LIN {X 0,Y 312.586,Z 149.548,A -85,B 0,C 180,E1 -15727.528,E2 -15727.528} C_VEL
LIN {X 0,Y 312.581,Z 149.547,A -85,B 0,C 180,E1 -15731.652,E2 -15731.652} C_VEL
LIN {X 0,Y 312.684,Z 149.533,A -85,B 0,C 180,E1 -15735.685,E2 -15735.685} C_VEL
LIN {X 0,Y 312.7,Z 149.532,A -85,B 0,C 180,E1 -15739.641,E2 -15739.641} C_VEL
LIN {X 0,Y 312.864,Z 149.511,A -85,B 0,C 180,E1 -15742.254,E2 -15742.254} C_VEL
LIN {X 0,Y 312.715,Z 149.533,A -85,B 0,C 180,E1 -15744.842,E2 -15744.842} C_VEL
LIN {X 0,Y 312.989,Z 149.499,A -85,B 0,C 180,E1 -15748.713,E2 -15748.713} C_VEL
LIN {X 0,Y 312.989,Z 149.496,A -85,B 0,C 180,E1 -15751.286,E2 -15751.286} C_VEL
LIN {X 0,Y 312.714,Z 149.531,A -85,B 0,C 180,E1 -15755.157,E2 -15755.157} C_VEL
LIN {X 0,Y 312.864,Z 149.51,A -85,B 0,C 180,E1 -15757.745,E2 -15757.745} C_VEL
LIN {X 0,Y 312.667,Z 149.535,A -85,B 0,C 180,E1 -15761.671,E2 -15761.671} C_VEL
LIN {X 0,Y 312.697,Z 149.533,A -85,B 0,C 180,E1 -15764.887,E2 -15764.887} C_VEL
LIN {X 0,Y 312.627,Z 149.54,A -85,B 0,C 180,E1 -15769.236,E2 -15769.236} C_VEL
LIN {X 0,Y 312.523,Z 149.554,A -85,B 0,C 180,E1 -15772.78,E2 -15772.78} C_VEL
LIN {X 0,Y 312.6,Z 149.546,A -85,B 0,C 180,E1 -15775.935,E2 -15775.935} C_VEL
LIN {X 0,Y 312.547,Z 149.551,A -85,B 0,C 180,E1 -15779.649,E2 -15779.649} C_VEL
LIN {X 0,Y 312.517,Z 149.556,A -85,B 0,C 180,E1 -15783.689,E2 -15783.689} C_VEL
LIN {X 0,Y 312.548,Z 149.55,A -85,B 0,C 180,E1 -15787.381,E2 -15787.381} C_VEL
LIN {X 0,Y 312.522,Z 149.553,A -85,B 0,C 180,E1 -15790.703,E2 -15790.703} C_VEL
LIN {X 0,Y 312.532,Z 149.554,A -85,B 0,C 180,E1 -15794.194,E2 -15794.194} C_VEL
LIN {X 0,Y 312.53,Z 149.556,A -85,B 0,C 180,E1 -15797.909,E2 -15797.909} C_VEL
LIN {X 0,Y 312.489,Z 149.557,A -85,B 0,C 180,E1 -15798.967,E2 -15798.967} C_VEL
LIN {X 0,Y 311.836,Z 149.643,A -85,B 0,C 180,E1 -15800.042,E2 -15800.042} C_VEL
LIN {X 0,Y 308.983,Z 149.998,A -85,B 0,C 180,E1 -15801.792,E2 -15801.792} C_VEL
LIN {X 0,Y 306.563,Z 150.296,A -85,B 0,C 180,E1 -15803.211,E2 -15803.211} C_VEL
LIN {X 0,Y 305.533,Z 150.424,A -85,B 0,C 180,E1 -15804.31,E2 -15804.31} C_VEL
LIN {X 0,Y 305.455,Z 150.433,A -85,B 0,C 180,E1 -15804.682,E2 -15804.682} C_VEL
LIN {X 0,Y 305.449,Z 150.434,A -85,B 0,C 180,E1 -15808.355,E2 -15808.355} C_VEL
LIN {X 0,Y 305.517,Z 150.427,A -85,B 0,C 180,E1 -15811.114,E2 -15811.114} C_VEL
LIN {X 0,Y 305.569,Z 150.42,A -85,B 0,C 180,E1 -15814.088,E2 -15814.088} C_VEL
LIN {X 0,Y 305.498,Z 150.428,A -85,B 0,C 180,E1 -15818.403,E2 -15818.403} C_VEL
LIN {X 0,Y 305.587,Z 150.421,A -85,B 0,C 180,E1 -15821.218,E2 -15821.218} C_VEL
LIN {X 0,Y 305.646,Z 150.413,A -85,B 0,C 180,E1 -15825.349,E2 -15825.349} C_VEL
LIN {X 0,Y 305.636,Z 150.413,A -85,B 0,C 180,E1 -15829.4,E2 -15829.4} C_VEL
LIN {X 0,Y 305.805,Z 150.39,A -85,B 0,C 180,E1 -15832.075,E2 -15832.075} C_VEL
LIN {X 0,Y 305.685,Z 150.407,A -85,B 0,C 180,E1 -15834.724,E2 -15834.724} C_VEL
LIN {X 0,Y 305.955,Z 150.374,A -85,B 0,C 180,E1 -15838.684,E2 -15838.684} C_VEL
LIN {X 0,Y 305.955,Z 150.372,A -85,B 0,C 180,E1 -15841.317,E2 -15841.317} C_VEL
LIN {X 0,Y 305.851,Z 150.388,A -85,B 0,C 180,E1 -15846.598,E2 -15846.598} C_VEL
LIN {X 0,Y 305.734,Z 150.399,A -85,B 0,C 180,E1 -15849.26,E2 -15849.26} C_VEL
LIN {X 0,Y 305.587,Z 150.417,A -85,B 0,C 180,E1 -15853.297,E2 -15853.297} C_VEL
LIN {X 0,Y 305.592,Z 150.418,A -85,B 0,C 180,E1 -15856.021,E2 -15856.021} C_VEL
LIN {X 0,Y 305.574,Z 150.418,A -85,B 0,C 180,E1 -15859.445,E2 -15859.445} C_VEL
LIN {X 0,Y 305.485,Z 150.43,A -85,B 0,C 180,E1 -15863.04,E2 -15863.04} C_VEL
LIN {X 0,Y 305.546,Z 150.427,A -85,B 0,C 180,E1 -15866.228,E2 -15866.228} C_VEL
LIN {X 0,Y 305.494,Z 150.428,A -85,B 0,C 180,E1 -15869.05,E2 -15869.05} C_VEL
LIN {X 0,Y 305.444,Z 150.438,A -85,B 0,C 180,E1 -15871.953,E2 -15871.953} C_VEL
LIN {X 0,Y 305.462,Z 150.432,A -85,B 0,C 180,E1 -15875.114,E2 -15875.114} C_VEL
LIN {X 0,Y 305.491,Z 150.43,A -85,B 0,C 180,E1 -15878.539,E2 -15878.539} C_VEL
LIN {X 0,Y 305.487,Z 150.43,A -85,B 0,C 180,E1 -15882.593,E2 -15882.593} C_VEL
LIN {X 0,Y 305.455,Z 150.435,A -85,B 0,C 180,E1 -15887.415,E2 -15887.415} C_VEL
LIN {X 0,Y 305.495,Z 150.432,A -85,B 0,C 180,E1 -15891.601,E2 -15891.601} C_VEL
LIN {X 0,Y 305.463,Z 150.433,A -85,B 0,C 180,E1 -15894.888,E2 -15894.888} C_VEL
LIN {X 0,Y 305.55,Z 150.588,A -85,B 0,C 180,E1 -15897.477,E2 -15897.477} C_VEL
LIN {X 0,Y 308.465,Z 164.645,A -85,B 0,C 180,E1 -15901.416,E2 -15901.416} C_VEL
LIN {X 0,Y 309.56,Z 170.48,A -85,B 0,C 180,E1 -15902.996,E2 -15902.996} C_VEL
LIN {X 0,Y 308.697,Z 179.088,A -85,B 0,C 180,E1 -15905.163,E2 -15905.163} C_VEL
LIN {X 0,Y 308.342,Z 181.983,A -85,B 0,C 180,E1 -15905.888,E2 -15905.888} C_VEL
LIN {X 0,Y 313.318,Z 226.374,A -85,B 0,C 180,E1 -15907.499,E2 -15907.499} C_VEL
LIN {X 0,Y 311.457,Z 291.139,A -85,B 0,C 180,E1 -15909.356,E2 -15909.356} C_VEL
LIN {X 0,Y 310.662,Z 304.701,A -85,B 0,C 180,E1 -15909.992,E2 -15909.992} C_VEL
LIN {X 0,Y 309.749,Z 316.693,A -85,B 0,C 180,E1 -15910.793,E2 -15910.793} C_VEL
LIN {X 0,Y 308.728,Z 327.693,A -85,B 0,C 180,E1 -15911.76,E2 -15911.76} C_VEL
LIN {X 0,Y 307.59,Z 339.295,A -85,B 0,C 180,E1 -15913.064,E2 -15913.064} C_VEL
LIN {X 0,Y 306.378,Z 350.376,A -85,B 0,C 180,E1 -15914.625,E2 -15914.625} C_VEL
LIN {X 0,Y 305.692,Z 358.469,A -85,B 0,C 180,E1 -15916.031,E2 -15916.031} C_VEL
LIN {X 0,Y 304.992,Z 366.419,A -85,B 0,C 180,E1 -15917.694,E2 -15917.694} C_VEL
LIN {X 0,Y 304.325,Z 374.155,A -85,B 0,C 180,E1 -15919.69,E2 -15919.69} C_VEL
LIN {X 0,Y 303.952,Z 381.267,A -85,B 0,C 180,E1 -15922.026,E2 -15922.026} C_VEL
LIN {X 0,Y 303.888,Z 385.785,A -85,B 0,C 180,E1 -15923.969,E2 -15923.969} C_VEL
LIN {X 0,Y 303.826,Z 389.338,A -85,B 0,C 180,E1 -15926.021,E2 -15926.021} C_VEL
LIN {X 0,Y 303.804,Z 391.012,A -85,B 0,C 180,E1 -15927.349,E2 -15927.349} C_VEL
LIN {X 0,Y 303.916,Z 392.26,A -85,B 0,C 180,E1 -15928.675,E2 -15928.675} C_VEL
LIN {X 0,Y 303.999,Z 393.067,A -85,B 0,C 180,E1 -15930,E2 -15930} C_VEL
LIN {X 0,Y 303.786,Z 393.382,A -85,B 0,C 180,E1 -15931.326,E2 -15931.326} C_VEL
LIN {X 0,Y 303.704,Z 393.287,A -85,B 0,C 180,E1 -15932.653,E2 -15932.653} C_VEL
LIN {X 0,Y 303.673,Z 392.784,A -85,B 0,C 180,E1 -15933.982,E2 -15933.982} C_VEL
LIN {X 0,Y 303.622,Z 391.636,A -85,B 0,C 180,E1 -15935.535,E2 -15935.535} C_VEL
LIN {X 0,Y 303.89,Z 388.673,A -85,B 0,C 180,E1 -15937.977,E2 -15937.977} C_VEL
LIN {X 0,Y 304.339,Z 385.131,A -85,B 0,C 180,E1 -15939.974,E2 -15939.974} C_VEL
LIN {X 0,Y 305.062,Z 380.498,A -85,B 0,C 180,E1 -15941.967,E2 -15941.967} C_VEL
LIN {X 0,Y 306.318,Z 374.653,A -85,B 0,C 180,E1 -15943.94,E2 -15943.94} C_VEL
LIN {X 0,Y 307.699,Z 367.423,A -85,B 0,C 180,E1 -15945.908,E2 -15945.908} C_VEL
LIN {X 0,Y 309.499,Z 358.5,A -85,B 0,C 180,E1 -15947.852,E2 -15947.852} C_VEL
LIN {X 0,Y 311.691,Z 348.451,A -85,B 0,C 180,E1 -15949.597,E2 -15949.597} C_VEL
LIN {X 0,Y 313.649,Z 338.405,A -85,B 0,C 180,E1 -15951.009,E2 -15951.009} C_VEL
LIN {X 0,Y 315.856,Z 325.87,A -85,B 0,C 180,E1 -15952.399,E2 -15952.399} C_VEL
LIN {X 0,Y 317.793,Z 313.439,A -85,B 0,C 180,E1 -15953.458,E2 -15953.458} C_VEL
LIN {X 0,Y 319.689,Z 299.024,A -85,B 0,C 180,E1 -15954.343,E2 -15954.343} C_VEL
LIN {X 0,Y 320.87,Z 286.162,A -85,B 0,C 180,E1 -15954.895,E2 -15954.895} C_VEL
LIN {X 0,Y 323.854,Z 227.495,A -85,B 0,C 180,E1 -15956.665,E2 -15956.665} C_VEL
LIN {X 0,Y 321.919,Z 211.124,A -85,B 0,C 180,E1 -15957.543,E2 -15957.543} C_VEL
LIN {X 0,Y 318.859,Z 193.947,A -85,B 0,C 180,E1 -15958.666,E2 -15958.666} C_VEL
LIN {X 0,Y 316.887,Z 185.521,A -85,B 0,C 180,E1 -15959.309,E2 -15959.309} C_VEL
LIN {X 0,Y 312.468,Z 176.034,A -85,B 0,C 180,E1 -15960.478,E2 -15960.478} C_VEL
LIN {X 0,Y 310.717,Z 168.166,A -85,B 0,C 180,E1 -15963.186,E2 -15963.186} C_VEL
LIN {X 0,Y 308.492,Z 160.006,A -85,B 0,C 180,E1 -15966.323,E2 -15966.323} C_VEL
LIN {X 0,Y 306.173,Z 152.7,A -85,B 0,C 180,E1 -15969.543,E2 -15969.543} C_VEL
LIN {X 0,Y 305.471,Z 150.434,A -85,B 0,C 180,E1 -15970.656,E2 -15970.656} C_VEL
LIN {X 0,Y 305.403,Z 150.44,A -85,B 0,C 180,E1 -15974.489,E2 -15974.489} C_VEL
LIN {X 0,Y 305.444,Z 150.431,A -85,B 0,C 180,E1 -15978.143,E2 -15978.143} C_VEL
LIN {X 0,Y 305.498,Z 150.424,A -85,B 0,C 180,E1 -15981.6,E2 -15981.6} C_VEL
LIN {X 0,Y 305.466,Z 150.431,A -85,B 0,C 180,E1 -15984.887,E2 -15984.887} C_VEL
LIN {X 0,Y 305.452,Z 150.428,A -85,B 0,C 180,E1 -15988.356,E2 -15988.356} C_VEL
LIN {X 0,Y 305.516,Z 150.423,A -85,B 0,C 180,E1 -15991.113,E2 -15991.113} C_VEL
LIN {X 0,Y 305.569,Z 150.415,A -85,B 0,C 180,E1 -15994.087,E2 -15994.087} C_VEL
LIN {X 0,Y 305.503,Z 150.431,A -85,B 0,C 180,E1 -15998.403,E2 -15998.403} C_VEL
LIN {X 0,Y 305.561,Z 150.421,A -85,B 0,C 180,E1 -16001.215,E2 -16001.215} C_VEL
LIN {X 0,Y 305.629,Z 150.415,A -85,B 0,C 180,E1 -16005.348,E2 -16005.348} C_VEL
LIN {X 0,Y 305.627,Z 150.415,A -85,B 0,C 180,E1 -16009.399,E2 -16009.399} C_VEL
LIN {X 0,Y 305.79,Z 150.494,A -85,B 0,C 180,E1 -16011.554,E2 -16011.554} C_VEL
LIN {X 0,Y 307.2,Z 154.947,A -85,B 0,C 180,E1 -16013.679,E2 -16013.679} C_VEL
LIN {X 0,Y 316.902,Z 170.364,A -85,B 0,C 180,E1 -16016.087,E2 -16016.087} C_VEL
LIN {X 0,Y 321.984,Z 179.999,A -85,B 0,C 180,E1 -16017.261,E2 -16017.261} C_VEL
LIN {X 0,Y 325.624,Z 188.448,A -85,B 0,C 180,E1 -16018.116,E2 -16018.116} C_VEL
LIN {X 0,Y 321.592,Z 261.751,A -85,B 0,C 180,E1 -16020.352,E2 -16020.352} C_VEL
LIN {X 0,Y 320.606,Z 274.961,A -85,B 0,C 180,E1 -16021.02,E2 -16021.02} C_VEL
LIN {X 0,Y 319.262,Z 287.316,A -85,B 0,C 180,E1 -16021.892,E2 -16021.892} C_VEL
LIN {X 0,Y 317.513,Z 299.966,A -85,B 0,C 180,E1 -16023.072,E2 -16023.072} C_VEL
LIN {X 0,Y 315.758,Z 310.435,A -85,B 0,C 180,E1 -16024.308,E2 -16024.308} C_VEL
LIN {X 0,Y 313.916,Z 320.373,A -85,B 0,C 180,E1 -16025.782,E2 -16025.782} C_VEL
LIN {X 0,Y 311.923,Z 329.891,A -85,B 0,C 180,E1 -16027.529,E2 -16027.529} C_VEL
LIN {X 0,Y 310.045,Z 338.248,A -85,B 0,C 180,E1 -16029.458,E2 -16029.458} C_VEL
LIN {X 0,Y 308.375,Z 345.16,A -85,B 0,C 180,E1 -16031.48,E2 -16031.48} C_VEL
LIN {X 0,Y 307.168,Z 349.957,A -85,B 0,C 180,E1 -16033.226,E2 -16033.226} C_VEL
LIN {X 0,Y 306.047,Z 354.407,A -85,B 0,C 180,E1 -16035.316,E2 -16035.316} C_VEL
LIN {X 0,Y 305.11,Z 357.667,A -85,B 0,C 180,E1 -16037.424,E2 -16037.424} C_VEL
LIN {X 0,Y 304.6,Z 359.297,A -85,B 0,C 180,E1 -16038.916,E2 -16038.916} C_VEL
LIN {X 0,Y 304.273,Z 360.262,A -85,B 0,C 180,E1 -16040.271,E2 -16040.271} C_VEL
LIN {X 0,Y 303.896,Z 360.929,A -85,B 0,C 180,E1 -16042.323,E2 -16042.323} C_VEL
LIN {X 0,Y 303.666,Z 360.491,A -85,B 0,C 180,E1 -16044.619,E2 -16044.619} C_VEL
LIN {X 0,Y 303.624,Z 359.576,A -85,B 0,C 180,E1 -16046.09,E2 -16046.09} C_VEL
LIN {X 0,Y 303.797,Z 356.925,A -85,B 0,C 180,E1 -16048.467,E2 -16048.467} C_VEL
LIN {X 0,Y 304.109,Z 353.399,A -85,B 0,C 180,E1 -16050.558,E2 -16050.558} C_VEL
LIN {X 0,Y 304.506,Z 348.138,A -85,B 0,C 180,E1 -16052.845,E2 -16052.845} C_VEL
LIN {X 0,Y 305.044,Z 342.283,A -85,B 0,C 180,E1 -16054.81,E2 -16054.81} C_VEL
LIN {X 0,Y 305.748,Z 335.246,A -85,B 0,C 180,E1 -16056.701,E2 -16056.701} C_VEL
LIN {X 0,Y 306.594,Z 326.786,A -85,B 0,C 180,E1 -16058.54,E2 -16058.54} C_VEL
LIN {X 0,Y 307.492,Z 317.339,A -85,B 0,C 180,E1 -16060.216,E2 -16060.216} C_VEL
LIN {X 0,Y 308.56,Z 306.406,A -85,B 0,C 180,E1 -16061.775,E2 -16061.775} C_VEL
LIN {X 0,Y 309.658,Z 293.744,A -85,B 0,C 180,E1 -16063.201,E2 -16063.201} C_VEL
LIN {X 0,Y 310.574,Z 280.985,A -85,B 0,C 180,E1 -16064.296,E2 -16064.296} C_VEL
LIN {X 0,Y 311.25,Z 267.383,A -85,B 0,C 180,E1 -16065.163,E2 -16065.163} C_VEL
LIN {X 0,Y 311.845,Z 253.446,A -85,B 0,C 180,E1 -16065.74,E2 -16065.74} C_VEL
LIN {X 0,Y 314.157,Z 176.783,A -85,B 0,C 180,E1 -16067.904,E2 -16067.904} C_VEL
LIN {X 0,Y 306.93,Z 154.768,A -85,B 0,C 180,E1 -16068.975,E2 -16068.975} C_VEL
LIN {X 0,Y 305.484,Z 150.432,A -85,B 0,C 180,E1 -16069.204,E2 -16069.204} C_VEL
LIN {X 0,Y 305.474,Z 150.434,A -85,B 0,C 180,E1 -16073.26,E2 -16073.26} C_VEL
LIN {X 0,Y 305.464,Z 150.432,A -85,B 0,C 180,E1 -16076.483,E2 -16076.483} C_VEL
LIN {X 0,Y 305.495,Z 150.43,A -85,B 0,C 180,E1 -16080.949,E2 -16080.949} C_VEL
LIN {X 0,Y 305.571,Z 150.419,A -85,B 0,C 180,E1 -16084.087,E2 -16084.087} C_VEL
LIN {X 0,Y 305.493,Z 150.429,A -85,B 0,C 180,E1 -16088.402,E2 -16088.402} C_VEL
LIN {X 0,Y 305.542,Z 150.428,A -85,B 0,C 180,E1 -16091.214,E2 -16091.214} C_VEL
LIN {X 0,Y 305.625,Z 150.415,A -85,B 0,C 180,E1 -16095.347,E2 -16095.347} C_VEL
LIN {X 0,Y 305.637,Z 150.413,A -85,B 0,C 180,E1 -16099.399,E2 -16099.399} C_VEL
LIN {X 0,Y 305.807,Z 150.389,A -85,B 0,C 180,E1 -16102.074,E2 -16102.074} C_VEL
LIN {X 0,Y 305.686,Z 150.408,A -85,B 0,C 180,E1 -16104.723,E2 -16104.723} C_VEL
LIN {X 0,Y 305.956,Z 150.375,A -85,B 0,C 180,E1 -16108.683,E2 -16108.683} C_VEL
LIN {X 0,Y 305.956,Z 150.372,A -85,B 0,C 180,E1 -16111.316,E2 -16111.316} C_VEL
LIN {X 0,Y 305.844,Z 150.39,A -85,B 0,C 180,E1 -16116.597,E2 -16116.597} C_VEL
LIN {X 0,Y 305.733,Z 150.399,A -85,B 0,C 180,E1 -16119.259,E2 -16119.259} C_VEL
LIN {X 0,Y 305.587,Z 150.417,A -85,B 0,C 180,E1 -16123.296,E2 -16123.296} C_VEL
LIN {X 0,Y 305.591,Z 150.418,A -85,B 0,C 180,E1 -16126.02,E2 -16126.02} C_VEL
LIN {X 0,Y 305.573,Z 150.418,A -85,B 0,C 180,E1 -16129.444,E2 -16129.444} C_VEL
LIN {X 0,Y 305.483,Z 150.43,A -85,B 0,C 180,E1 -16133.039,E2 -16133.039} C_VEL
LIN {X 0,Y 305.545,Z 150.427,A -85,B 0,C 180,E1 -16136.227,E2 -16136.227} C_VEL
LIN {X 0,Y 305.501,Z 150.427,A -85,B 0,C 180,E1 -16139.052,E2 -16139.052} C_VEL
LIN {X 0,Y 305.445,Z 150.438,A -85,B 0,C 180,E1 -16141.951,E2 -16141.951} C_VEL
LIN {X 0,Y 305.459,Z 150.432,A -85,B 0,C 180,E1 -16145.113,E2 -16145.113} C_VEL
LIN {X 0,Y 305.489,Z 150.43,A -85,B 0,C 180,E1 -16148.539,E2 -16148.539} C_VEL
LIN {X 0,Y 305.506,Z 150.427,A -85,B 0,C 180,E1 -16152.597,E2 -16152.597} C_VEL
LIN {X 0,Y 305.484,Z 150.431,A -85,B 0,C 180,E1 -16156.356,E2 -16156.356} C_VEL
LIN {X 0,Y 305.462,Z 150.436,A -85,B 0,C 180,E1 -16159.894,E2 -16159.894} C_VEL
LIN {X 0,Y 305.496,Z 150.433,A -85,B 0,C 180,E1 -16163.627,E2 -16163.627} C_VEL
LIN {X 0,Y 305.455,Z 150.433,A -85,B 0,C 180,E1 -16164.682,E2 -16164.682} C_VEL
LIN {X 0,Y 304.794,Z 150.519,A -85,B 0,C 180,E1 -16165.783,E2 -16165.783} C_VEL
LIN {X 0,Y 301.922,Z 150.879,A -85,B 0,C 180,E1 -16167.575,E2 -16167.575} C_VEL
LIN {X 0,Y 299.5,Z 151.177,A -85,B 0,C 180,E1 -16169.028,E2 -16169.028} C_VEL
LIN {X 0,Y 298.49,Z 151.302,A -85,B 0,C 180,E1 -16170.154,E2 -16170.154} C_VEL
LIN {X 0,Y 298.425,Z 151.308,A -85,B 0,C 180,E1 -16170.536,E2 -16170.536} C_VEL
LIN {X 0,Y 298.489,Z 151.306,A -85,B 0,C 180,E1 -16173.471,E2 -16173.471} C_VEL
LIN {X 0,Y 298.432,Z 151.309,A -85,B 0,C 180,E1 -16176.698,E2 -16176.698} C_VEL
LIN {X 0,Y 298.537,Z 151.296,A -85,B 0,C 180,E1 -16180.757,E2 -16180.757} C_VEL
LIN {X 0,Y 298.591,Z 151.292,A -85,B 0,C 180,E1 -16184.995,E2 -16184.995} C_VEL
LIN {X 0,Y 298.591,Z 151.293,A -85,B 0,C 180,E1 -16189.147,E2 -16189.147} C_VEL
LIN {X 0,Y 298.752,Z 151.268,A -85,B 0,C 180,E1 -16191.886,E2 -16191.886} C_VEL
LIN {X 0,Y 298.656,Z 151.282,A -85,B 0,C 180,E1 -16194.599,E2 -16194.599} C_VEL
LIN {X 0,Y 298.922,Z 151.25,A -85,B 0,C 180,E1 -16198.653,E2 -16198.653} C_VEL
LIN {X 0,Y 298.922,Z 151.248,A -85,B 0,C 180,E1 -16201.348,E2 -16201.348} C_VEL
LIN {X 0,Y 298.796,Z 151.268,A -85,B 0,C 180,E1 -16206.754,E2 -16206.754} C_VEL
LIN {X 0,Y 298.679,Z 151.278,A -85,B 0,C 180,E1 -16209.481,E2 -16209.481} C_VEL
LIN {X 0,Y 298.551,Z 151.293,A -85,B 0,C 180,E1 -16213.616,E2 -16213.616} C_VEL
LIN {X 0,Y 298.547,Z 151.298,A -85,B 0,C 180,E1 -16216.409,E2 -16216.409} C_VEL
LIN {X 0,Y 298.509,Z 151.298,A -85,B 0,C 180,E1 -16219.655,E2 -16219.655} C_VEL
LIN {X 0,Y 298.427,Z 151.309,A -85,B 0,C 180,E1 -16223.601,E2 -16223.601} C_VEL
LIN {X 0,Y 298.488,Z 151.304,A -85,B 0,C 180,E1 -16226.575,E2 -16226.575} C_VEL
LIN {X 0,Y 298.42,Z 151.31,A -85,B 0,C 180,E1 -16229.642,E2 -16229.642} C_VEL
LIN {X 0,Y 298.395,Z 151.314,A -85,B 0,C 180,E1 -16232.801,E2 -16232.801} C_VEL
LIN {X 0,Y 298.47,Z 151.303,A -85,B 0,C 180,E1 -16236.814,E2 -16236.814} C_VEL
LIN {X 0,Y 298.418,Z 151.31,A -85,B 0,C 180,E1 -16241.095,E2 -16241.095} C_VEL
LIN {X 0,Y 298.426,Z 151.309,A -85,B 0,C 180,E1 -16243.11,E2 -16243.11} C_VEL
LIN {X 0,Y 298.403,Z 151.312,A -85,B 0,C 180,E1 -16246.922,E2 -16246.922} C_VEL
LIN {X 0,Y 298.415,Z 151.311,A -85,B 0,C 180,E1 -16251.004,E2 -16251.004} C_VEL
LIN {X 0,Y 298.419,Z 151.314,A -85,B 0,C 180,E1 -16253.931,E2 -16253.931} C_VEL
LIN {X 0,Y 298.471,Z 151.352,A -85,B 0,C 180,E1 -16257.16,E2 -16257.16} C_VEL
LIN {X 0,Y 301.311,Z 164.922,A -85,B 0,C 180,E1 -16261.055,E2 -16261.055} C_VEL
LIN {X 0,Y 302.563,Z 172.208,A -85,B 0,C 180,E1 -16263.067,E2 -16263.067} C_VEL
LIN {X 0,Y 301.467,Z 181.646,A -85,B 0,C 180,E1 -16265.49,E2 -16265.49} C_VEL
LIN {X 0,Y 306.452,Z 226.423,A -85,B 0,C 180,E1 -16267.167,E2 -16267.167} C_VEL
LIN {X 0,Y 304.508,Z 291.26,A -85,B 0,C 180,E1 -16269.083,E2 -16269.083} C_VEL
LIN {X 0,Y 303.666,Z 305.37,A -85,B 0,C 180,E1 -16269.775,E2 -16269.775} C_VEL
LIN {X 0,Y 302.671,Z 318.042,A -85,B 0,C 180,E1 -16270.678,E2 -16270.678} C_VEL
LIN {X 0,Y 301.467,Z 330.243,A -85,B 0,C 180,E1 -16271.832,E2 -16271.832} C_VEL
LIN {X 0,Y 300.379,Z 341.324,A -85,B 0,C 180,E1 -16273.17,E2 -16273.17} C_VEL
LIN {X 0,Y 299.19,Z 351.635,A -85,B 0,C 180,E1 -16274.731,E2 -16274.731} C_VEL
LIN {X 0,Y 298.554,Z 358.819,A -85,B 0,C 180,E1 -16276.038,E2 -16276.038} C_VEL
LIN {X 0,Y 297.854,Z 366.641,A -85,B 0,C 180,E1 -16277.74,E2 -16277.74} C_VEL
LIN {X 0,Y 297.231,Z 374.28,A -85,B 0,C 180,E1 -16279.786,E2 -16279.786} C_VEL
LIN {X 0,Y 296.902,Z 380.38,A -85,B 0,C 180,E1 -16281.835,E2 -16281.835} C_VEL
LIN {X 0,Y 296.803,Z 385.375,A -85,B 0,C 180,E1 -16284.003,E2 -16284.003} C_VEL
LIN {X 0,Y 296.764,Z 388.686,A -85,B 0,C 180,E1 -16285.926,E2 -16285.926} C_VEL
LIN {X 0,Y 296.723,Z 390.414,A -85,B 0,C 180,E1 -16287.285,E2 -16287.285} C_VEL
LIN {X 0,Y 296.826,Z 391.706,A -85,B 0,C 180,E1 -16288.644,E2 -16288.644} C_VEL
LIN {X 0,Y 296.924,Z 392.569,A -85,B 0,C 180,E1 -16290.001,E2 -16290.001} C_VEL
LIN {X 0,Y 296.694,Z 392.955,A -85,B 0,C 180,E1 -16291.358,E2 -16291.358} C_VEL
LIN {X 0,Y 296.623,Z 392.901,A -85,B 0,C 180,E1 -16292.717,E2 -16292.717} C_VEL
LIN {X 0,Y 296.583,Z 392.441,A -85,B 0,C 180,E1 -16294.077,E2 -16294.077} C_VEL
LIN {X 0,Y 296.548,Z 391.522,A -85,B 0,C 180,E1 -16295.509,E2 -16295.509} C_VEL
LIN {X 0,Y 296.618,Z 390.264,A -85,B 0,C 180,E1 -16296.804,E2 -16296.804} C_VEL
LIN {X 0,Y 296.985,Z 387.5,A -85,B 0,C 180,E1 -16298.849,E2 -16298.849} C_VEL
LIN {X 0,Y 297.57,Z 383.699,A -85,B 0,C 180,E1 -16300.892,E2 -16300.892} C_VEL
LIN {X 0,Y 298.496,Z 378.775,A -85,B 0,C 180,E1 -16302.925,E2 -16302.925} C_VEL
LIN {X 0,Y 300.168,Z 371.468,A -85,B 0,C 180,E1 -16305.273,E2 -16305.273} C_VEL
LIN {X 0,Y 301.753,Z 363.674,A -85,B 0,C 180,E1 -16307.269,E2 -16307.269} C_VEL
LIN {X 0,Y 303.573,Z 355.722,A -85,B 0,C 180,E1 -16308.912,E2 -16308.912} C_VEL
LIN {X 0,Y 305.828,Z 345.069,A -85,B 0,C 180,E1 -16310.691,E2 -16310.691} C_VEL
LIN {X 0,Y 308.146,Z 334.358,A -85,B 0,C 180,E1 -16312.106,E2 -16312.106} C_VEL
LIN {X 0,Y 310.222,Z 322.647,A -85,B 0,C 180,E1 -16313.357,E2 -16313.357} C_VEL
LIN {X 0,Y 312.367,Z 309.416,A -85,B 0,C 180,E1 -16314.42,E2 -16314.42} C_VEL
LIN {X 0,Y 314.102,Z 295.961,A -85,B 0,C 180,E1 -16315.203,E2 -16315.203} C_VEL
LIN {X 0,Y 315.278,Z 281.766,A -85,B 0,C 180,E1 -16315.766,E2 -16315.766} C_VEL
LIN {X 0,Y 318.146,Z 228.588,A -85,B 0,C 180,E1 -16317.391,E2 -16317.391} C_VEL
LIN {X 0,Y 316.306,Z 212.407,A -85,B 0,C 180,E1 -16318.305,E2 -16318.305} C_VEL
LIN {X 0,Y 313.5,Z 196.283,A -85,B 0,C 180,E1 -16319.397,E2 -16319.397} C_VEL
LIN {X 0,Y 311.853,Z 189.166,A -85,B 0,C 180,E1 -16319.968,E2 -16319.968} C_VEL
LIN {X 0,Y 307.38,Z 179.825,A -85,B 0,C 180,E1 -16321.16,E2 -16321.16} C_VEL
LIN {X 0,Y 305.28,Z 175.365,A -85,B 0,C 180,E1 -16321.792,E2 -16321.792} C_VEL
LIN {X 0,Y 303.469,Z 167.901,A -85,B 0,C 180,E1 -16324.569,E2 -16324.569} C_VEL
LIN {X 0,Y 301.456,Z 160.696,A -85,B 0,C 180,E1 -16327.564,E2 -16327.564} C_VEL
LIN {X 0,Y 299.567,Z 154.906,A -85,B 0,C 180,E1 -16330.318,E2 -16330.318} C_VEL
LIN {X 0,Y 298.424,Z 151.31,A -85,B 0,C 180,E1 -16332.262,E2 -16332.262} C_VEL
LIN {X 0,Y 298.406,Z 151.311,A -85,B 0,C 180,E1 -16336.921,E2 -16336.921} C_VEL
LIN {X 0,Y 298.418,Z 151.303,A -85,B 0,C 180,E1 -16341.004,E2 -16341.004} C_VEL
LIN {X 0,Y 298.424,Z 151.303,A -85,B 0,C 180,E1 -16343.93,E2 -16343.93} C_VEL
LIN {X 0,Y 298.397,Z 151.309,A -85,B 0,C 180,E1 -16347.984,E2 -16347.984} C_VEL
LIN {X 0,Y 298.461,Z 151.302,A -85,B 0,C 180,E1 -16351.903,E2 -16351.903} C_VEL
LIN {X 0,Y 298.487,Z 151.3,A -85,B 0,C 180,E1 -16354.924,E2 -16354.924} C_VEL
LIN {X 0,Y 298.45,Z 151.303,A -85,B 0,C 180,E1 -16359.315,E2 -16359.315} C_VEL
LIN {X 0,Y 298.512,Z 151.295,A -85,B 0,C 180,E1 -16362.177,E2 -16362.177} C_VEL
LIN {X 0,Y 298.589,Z 151.288,A -85,B 0,C 180,E1 -16364.994,E2 -16364.994} C_VEL
LIN {X 0,Y 298.586,Z 151.29,A -85,B 0,C 180,E1 -16369.146,E2 -16369.146} C_VEL
LIN {X 0,Y 298.617,Z 151.462,A -85,B 0,C 180,E1 -16370.004,E2 -16370.004} C_VEL
LIN {X 0,Y 300.196,Z 155.742,A -85,B 0,C 180,E1 -16372.284,E2 -16372.284} C_VEL
LIN {X 0,Y 304.459,Z 162.336,A -85,B 0,C 180,E1 -16373.499,E2 -16373.499} C_VEL
LIN {X 0,Y 312.551,Z 175.162,A -85,B 0,C 180,E1 -16375.566,E2 -16375.566} C_VEL
LIN {X 0,Y 317.309,Z 184.427,A -85,B 0,C 180,E1 -16376.728,E2 -16376.728} C_VEL
LIN {X 0,Y 320.036,Z 190.794,A -85,B 0,C 180,E1 -16377.401,E2 -16377.401} C_VEL
LIN {X 0,Y 315.811,Z 261.792,A -85,B 0,C 180,E1 -16379.613,E2 -16379.613} C_VEL
LIN {X 0,Y 314.792,Z 274.33,A -85,B 0,C 180,E1 -16380.239,E2 -16380.239} C_VEL
LIN {X 0,Y 313.442,Z 286.936,A -85,B 0,C 180,E1 -16381.124,E2 -16381.124} C_VEL
LIN {X 0,Y 311.646,Z 299.174,A -85,B 0,C 180,E1 -16382.261,E2 -16382.261} C_VEL
LIN {X 0,Y 309.621,Z 310.675,A -85,B 0,C 180,E1 -16383.631,E2 -16383.631} C_VEL
LIN {X 0,Y 307.751,Z 320.284,A -85,B 0,C 180,E1 -16385.076,E2 -16385.076} C_VEL
LIN {X 0,Y 305.919,Z 328.628,A -85,B 0,C 180,E1 -16386.595,E2 -16386.595} C_VEL
LIN {X 0,Y 303.73,Z 337.727,A -85,B 0,C 180,E1 -16388.65,E2 -16388.65} C_VEL
LIN {X 0,Y 301.887,Z 344.926,A -85,B 0,C 180,E1 -16390.733,E2 -16390.733} C_VEL
LIN {X 0,Y 300.347,Z 350.607,A -85,B 0,C 180,E1 -16392.843,E2 -16392.843} C_VEL
LIN {X 0,Y 299.157,Z 354.976,A -85,B 0,C 180,E1 -16394.976,E2 -16394.976} C_VEL
LIN {X 0,Y 298.463,Z 357.275,A -85,B 0,C 180,E1 -16396.413,E2 -16396.413} C_VEL
LIN {X 0,Y 297.478,Z 360.119,A -85,B 0,C 180,E1 -16399.088,E2 -16399.088} C_VEL
LIN {X 0,Y 297.096,Z 361.081,A -85,B 0,C 180,E1 -16400.783,E2 -16400.783} C_VEL
LIN {X 0,Y 296.79,Z 361.374,A -85,B 0,C 180,E1 -16402.553,E2 -16402.553} C_VEL
LIN {X 0,Y 296.645,Z 361.183,A -85,B 0,C 180,E1 -16403.75,E2 -16403.75} C_VEL
LIN {X 0,Y 296.561,Z 360.099,A -85,B 0,C 180,E1 -16405.77,E2 -16405.77} C_VEL
LIN {X 0,Y 296.67,Z 357.453,A -85,B 0,C 180,E1 -16408.28,E2 -16408.28} C_VEL
LIN {X 0,Y 297.034,Z 353.67,A -85,B 0,C 180,E1 -16410.577,E2 -16410.577} C_VEL
LIN {X 0,Y 297.443,Z 348.367,A -85,B 0,C 180,E1 -16412.918,E2 -16412.918} C_VEL
LIN {X 0,Y 297.972,Z 342.594,A -85,B 0,C 180,E1 -16414.887,E2 -16414.887} C_VEL
LIN {X 0,Y 298.707,Z 335.306,A -85,B 0,C 180,E1 -16416.874,E2 -16416.874} C_VEL
LIN {X 0,Y 299.625,Z 326.238,A -85,B 0,C 180,E1 -16418.861,E2 -16418.861} C_VEL
LIN {X 0,Y 300.492,Z 317.509,A -85,B 0,C 180,E1 -16420.423,E2 -16420.423} C_VEL
LIN {X 0,Y 301.46,Z 308.031,A -85,B 0,C 180,E1 -16421.821,E2 -16421.821} C_VEL
LIN {X 0,Y 302.55,Z 295.876,A -85,B 0,C 180,E1 -16423.255,E2 -16423.255} C_VEL
LIN {X 0,Y 303.465,Z 284,A -85,B 0,C 180,E1 -16424.356,E2 -16424.356} C_VEL
LIN {X 0,Y 304.225,Z 270.889,A -85,B 0,C 180,E1 -16425.264,E2 -16425.264} C_VEL
LIN {X 0,Y 304.815,Z 256.905,A -85,B 0,C 180,E1 -16425.935,E2 -16425.935} C_VEL
LIN {X 0,Y 307.316,Z 177.999,A -85,B 0,C 180,E1 -16428.236,E2 -16428.236} C_VEL
LIN {X 0,Y 300.604,Z 157.594,A -85,B 0,C 180,E1 -16429.261,E2 -16429.261} C_VEL
LIN {X 0,Y 298.434,Z 151.313,A -85,B 0,C 180,E1 -16429.61,E2 -16429.61} C_VEL
LIN {X 0,Y 298.418,Z 151.313,A -85,B 0,C 180,E1 -16433.93,E2 -16433.93} C_VEL
LIN {X 0,Y 298.395,Z 151.315,A -85,B 0,C 180,E1 -16437.983,E2 -16437.983} C_VEL
LIN {X 0,Y 298.469,Z 151.306,A -85,B 0,C 180,E1 -16441.904,E2 -16441.904} C_VEL
LIN {X 0,Y 298.485,Z 151.304,A -85,B 0,C 180,E1 -16444.924,E2 -16444.924} C_VEL
LIN {X 0,Y 298.438,Z 151.312,A -85,B 0,C 180,E1 -16449.314,E2 -16449.314} C_VEL
LIN {X 0,Y 298.476,Z 151.303,A -85,B 0,C 180,E1 -16452.175,E2 -16452.175} C_VEL
LIN {X 0,Y 298.584,Z 151.293,A -85,B 0,C 180,E1 -16454.994,E2 -16454.994} C_VEL
LIN {X 0,Y 298.592,Z 151.293,A -85,B 0,C 180,E1 -16459.146,E2 -16459.146} C_VEL
LIN {X 0,Y 298.753,Z 151.268,A -85,B 0,C 180,E1 -16461.885,E2 -16461.885} C_VEL
LIN {X 0,Y 298.656,Z 151.282,A -85,B 0,C 180,E1 -16464.598,E2 -16464.598} C_VEL
LIN {X 0,Y 298.922,Z 151.251,A -85,B 0,C 180,E1 -16468.652,E2 -16468.652} C_VEL
LIN {X 0,Y 298.922,Z 151.248,A -85,B 0,C 180,E1 -16471.347,E2 -16471.347} C_VEL
LIN {X 0,Y 298.79,Z 151.268,A -85,B 0,C 180,E1 -16476.754,E2 -16476.754} C_VEL
LIN {X 0,Y 298.678,Z 151.277,A -85,B 0,C 180,E1 -16479.48,E2 -16479.48} C_VEL
LIN {X 0,Y 298.55,Z 151.293,A -85,B 0,C 180,E1 -16483.615,E2 -16483.615} C_VEL
LIN {X 0,Y 298.546,Z 151.299,A -85,B 0,C 180,E1 -16486.408,E2 -16486.408} C_VEL
LIN {X 0,Y 298.507,Z 151.298,A -85,B 0,C 180,E1 -16489.654,E2 -16489.654} C_VEL
LIN {X 0,Y 298.426,Z 151.309,A -85,B 0,C 180,E1 -16493.6,E2 -16493.6} C_VEL
LIN {X 0,Y 298.487,Z 151.303,A -85,B 0,C 180,E1 -16496.574,E2 -16496.574} C_VEL
LIN {X 0,Y 298.422,Z 151.31,A -85,B 0,C 180,E1 -16499.64,E2 -16499.64} C_VEL
LIN {X 0,Y 298.394,Z 151.313,A -85,B 0,C 180,E1 -16502.8,E2 -16502.8} C_VEL
LIN {X 0,Y 298.466,Z 151.304,A -85,B 0,C 180,E1 -16506.814,E2 -16506.814} C_VEL
LIN {X 0,Y 298.448,Z 151.307,A -85,B 0,C 180,E1 -16511.25,E2 -16511.25} C_VEL
LIN {X 0,Y 298.413,Z 151.31,A -85,B 0,C 180,E1 -16515.047,E2 -16515.047} C_VEL
LIN {X 0,Y 298.417,Z 151.31,A -85,B 0,C 180,E1 -16518.745,E2 -16518.745} C_VEL
LIN {X 0,Y 298.441,Z 151.307,A -85,B 0,C 180,E1 -16522.247,E2 -16522.247} C_VEL
LIN {X 0,Y 298.405,Z 151.316,A -85,B 0,C 180,E1 -16525.581,E2 -16525.581} C_VEL
LIN {X 0,Y 298.392,Z 151.313,A -85,B 0,C 180,E1 -16528.791,E2 -16528.791} C_VEL
LIN {X 0,Y 298.425,Z 151.308,A -85,B 0,C 180,E1 -16530.536,E2 -16530.536} C_VEL
LIN {X 0,Y 297.817,Z 151.388,A -85,B 0,C 180,E1 -16531.662,E2 -16531.662} C_VEL
LIN {X 0,Y 295.034,Z 151.736,A -85,B 0,C 180,E1 -16533.499,E2 -16533.499} C_VEL
LIN {X 0,Y 292.614,Z 152.035,A -85,B 0,C 180,E1 -16534.988,E2 -16534.988} C_VEL
LIN {X 0,Y 291.53,Z 152.169,A -85,B 0,C 180,E1 -16536.141,E2 -16536.141} C_VEL
LIN {X 0,Y 291.419,Z 152.182,A -85,B 0,C 180,E1 -16536.532,E2 -16536.532} C_VEL
LIN {X 0,Y 291.455,Z 152.177,A -85,B 0,C 180,E1 -16540.271,E2 -16540.271} C_VEL
LIN {X 0,Y 291.552,Z 152.166,A -85,B 0,C 180,E1 -16544.624,E2 -16544.624} C_VEL
LIN {X 0,Y 291.534,Z 152.17,A -85,B 0,C 180,E1 -16548.881,E2 -16548.881} C_VEL
LIN {X 0,Y 291.703,Z 152.147,A -85,B 0,C 180,E1 -16551.689,E2 -16551.689} C_VEL
LIN {X 0,Y 291.626,Z 152.157,A -85,B 0,C 180,E1 -16554.469,E2 -16554.469} C_VEL
LIN {X 0,Y 291.888,Z 152.126,A -85,B 0,C 180,E1 -16558.621,E2 -16558.621} C_VEL
LIN {X 0,Y 291.888,Z 152.124,A -85,B 0,C 180,E1 -16561.38,E2 -16561.38} C_VEL
LIN {X 0,Y 291.745,Z 152.145,A -85,B 0,C 180,E1 -16566.918,E2 -16566.918} C_VEL
LIN {X 0,Y 291.628,Z 152.156,A -85,B 0,C 180,E1 -16569.712,E2 -16569.712} C_VEL
LIN {X 0,Y 291.521,Z 152.169,A -85,B 0,C 180,E1 -16573.951,E2 -16573.951} C_VEL
LIN {X 0,Y 291.486,Z 152.176,A -85,B 0,C 180,E1 -16576.818,E2 -16576.818} C_VEL
LIN {X 0,Y 291.449,Z 152.178,A -85,B 0,C 180,E1 -16579.875,E2 -16579.875} C_VEL
LIN {X 0,Y 291.382,Z 152.19,A -85,B 0,C 180,E1 -16584.207,E2 -16584.207} C_VEL
LIN {X 0,Y 291.422,Z 152.181,A -85,B 0,C 180,E1 -16587.272,E2 -16587.272} C_VEL
LIN {X 0,Y 291.337,Z 152.195,A -85,B 0,C 180,E1 -16590.437,E2 -16590.437} C_VEL
LIN {X 0,Y 291.344,Z 152.193,A -85,B 0,C 180,E1 -16593.699,E2 -16593.699} C_VEL
LIN {X 0,Y 291.404,Z 152.183,A -85,B 0,C 180,E1 -16597.262,E2 -16597.262} C_VEL
LIN {X 0,Y 291.377,Z 152.188,A -85,B 0,C 180,E1 -16600.636,E2 -16600.636} C_VEL
LIN {X 0,Y 291.299,Z 152.197,A -85,B 0,C 180,E1 -16604.401,E2 -16604.401} C_VEL
LIN {X 0,Y 291.326,Z 152.195,A -85,B 0,C 180,E1 -16608.405,E2 -16608.405} C_VEL
LIN {X 0,Y 291.364,Z 152.19,A -85,B 0,C 180,E1 -16611.161,E2 -16611.161} C_VEL
LIN {X 0,Y 291.362,Z 152.19,A -85,B 0,C 180,E1 -16614.627,E2 -16614.627} C_VEL
LIN {X 0,Y 291.405,Z 152.279,A -85,B 0,C 180,E1 -16616.875,E2 -16616.875} C_VEL
LIN {X 0,Y 294.41,Z 166.621,A -85,B 0,C 180,E1 -16621.093,E2 -16621.093} C_VEL
LIN {X 0,Y 295.521,Z 172.532,A -85,B 0,C 180,E1 -16622.766,E2 -16622.766} C_VEL
LIN {X 0,Y 294.579,Z 181.534,A -85,B 0,C 180,E1 -16625.091,E2 -16625.091} C_VEL
LIN {X 0,Y 299.559,Z 227.691,A -85,B 0,C 180,E1 -16626.858,E2 -16626.858} C_VEL
LIN {X 0,Y 297.58,Z 291.39,A -85,B 0,C 180,E1 -16628.8,E2 -16628.8} C_VEL
LIN {X 0,Y 296.787,Z 304.621,A -85,B 0,C 180,E1 -16629.467,E2 -16629.467} C_VEL
LIN {X 0,Y 295.751,Z 317.396,A -85,B 0,C 180,E1 -16630.388,E2 -16630.388} C_VEL
LIN {X 0,Y 294.518,Z 329.644,A -85,B 0,C 180,E1 -16631.568,E2 -16631.568} C_VEL
LIN {X 0,Y 293.399,Z 340.773,A -85,B 0,C 180,E1 -16632.937,E2 -16632.937} C_VEL
LIN {X 0,Y 292.12,Z 351.812,A -85,B 0,C 180,E1 -16634.655,E2 -16634.655} C_VEL
LIN {X 0,Y 291.295,Z 360.841,A -85,B 0,C 180,E1 -16636.395,E2 -16636.395} C_VEL
LIN {X 0,Y 290.59,Z 368.262,A -85,B 0,C 180,E1 -16638.137,E2 -16638.137} C_VEL
LIN {X 0,Y 290.021,Z 375.495,A -85,B 0,C 180,E1 -16640.234,E2 -16640.234} C_VEL
LIN {X 0,Y 289.767,Z 381.234,A -85,B 0,C 180,E1 -16642.335,E2 -16642.335} C_VEL
LIN {X 0,Y 289.705,Z 385.676,A -85,B 0,C 180,E1 -16644.432,E2 -16644.432} C_VEL
LIN {X 0,Y 289.702,Z 387.989,A -85,B 0,C 180,E1 -16645.827,E2 -16645.827} C_VEL
LIN {X 0,Y 289.644,Z 389.804,A -85,B 0,C 180,E1 -16647.219,E2 -16647.219} C_VEL
LIN {X 0,Y 289.737,Z 391.138,A -85,B 0,C 180,E1 -16648.611,E2 -16648.611} C_VEL
LIN {X 0,Y 289.851,Z 392.046,A -85,B 0,C 180,E1 -16650.001,E2 -16650.001} C_VEL
LIN {X 0,Y 289.604,Z 392.506,A -85,B 0,C 180,E1 -16651.391,E2 -16651.391} C_VEL
LIN {X 0,Y 289.544,Z 392.517,A -85,B 0,C 180,E1 -16652.783,E2 -16652.783} C_VEL
LIN {X 0,Y 289.437,Z 391.397,A -85,B 0,C 180,E1 -16655.404,E2 -16655.404} C_VEL
LIN {X 0,Y 289.553,Z 390.051,A -85,B 0,C 180,E1 -16656.971,E2 -16656.971} C_VEL
LIN {X 0,Y 289.923,Z 387.362,A -85,B 0,C 180,E1 -16659.066,E2 -16659.066} C_VEL
LIN {X 0,Y 290.565,Z 383.674,A -85,B 0,C 180,E1 -16661.158,E2 -16661.158} C_VEL
LIN {X 0,Y 291.566,Z 378.898,A -85,B 0,C 180,E1 -16663.238,E2 -16663.238} C_VEL
LIN {X 0,Y 293.327,Z 371.748,A -85,B 0,C 180,E1 -16665.638,E2 -16665.638} C_VEL
LIN {X 0,Y 294.914,Z 364.443,A -85,B 0,C 180,E1 -16667.592,E2 -16667.592} C_VEL
LIN {X 0,Y 296.901,Z 356.311,A -85,B 0,C 180,E1 -16669.354,E2 -16669.354} C_VEL
LIN {X 0,Y 299.029,Z 347.079,A -85,B 0,C 180,E1 -16671.003,E2 -16671.003} C_VEL
LIN {X 0,Y 301.67,Z 335.665,A -85,B 0,C 180,E1 -16672.607,E2 -16672.607} C_VEL
LIN {X 0,Y 303.839,Z 324.392,A -85,B 0,C 180,E1 -16673.878,E2 -16673.878} C_VEL
LIN {X 0,Y 306.007,Z 311.87,A -85,B 0,C 180,E1 -16674.962,E2 -16674.962} C_VEL
LIN {X 0,Y 308.059,Z 297.428,A -85,B 0,C 180,E1 -16675.869,E2 -16675.869} C_VEL
LIN {X 0,Y 309.379,Z 283.198,A -85,B 0,C 180,E1 -16676.476,E2 -16676.476} C_VEL
LIN {X 0,Y 312.532,Z 229.371,A -85,B 0,C 180,E1 -16678.18,E2 -16678.18} C_VEL
LIN {X 0,Y 310.722,Z 213.529,A -85,B 0,C 180,E1 -16679.115,E2 -16679.115} C_VEL
LIN {X 0,Y 308.352,Z 199.12,A -85,B 0,C 180,E1 -16680.13,E2 -16680.13} C_VEL
LIN {X 0,Y 306.918,Z 192.788,A -85,B 0,C 180,E1 -16680.662,E2 -16680.662} C_VEL
LIN {X 0,Y 302.95,Z 184.33,A -85,B 0,C 180,E1 -16681.777,E2 -16681.777} C_VEL
LIN {X 0,Y 300.231,Z 179.012,A -85,B 0,C 180,E1 -16682.572,E2 -16682.572} C_VEL
LIN {X 0,Y 298.052,Z 174.602,A -85,B 0,C 180,E1 -16683.286,E2 -16683.286} C_VEL
LIN {X 0,Y 296.078,Z 166.936,A -85,B 0,C 180,E1 -16686.401,E2 -16686.401} C_VEL
LIN {X 0,Y 294.119,Z 160.44,A -85,B 0,C 180,E1 -16689.417,E2 -16689.417} C_VEL
LIN {X 0,Y 292.025,Z 154.353,A -85,B 0,C 180,E1 -16692.729,E2 -16692.729} C_VEL
LIN {X 0,Y 291.307,Z 152.195,A -85,B 0,C 180,E1 -16694.076,E2 -16694.076} C_VEL
LIN {X 0,Y 291.323,Z 152.195,A -85,B 0,C 180,E1 -16697.508,E2 -16697.508} C_VEL
LIN {X 0,Y 291.367,Z 152.181,A -85,B 0,C 180,E1 -16701.16,E2 -16701.16} C_VEL
LIN {X 0,Y 291.383,Z 152.185,A -85,B 0,C 180,E1 -16704.629,E2 -16704.629} C_VEL
LIN {X 0,Y 291.374,Z 152.184,A -85,B 0,C 180,E1 -16707.95,E2 -16707.95} C_VEL
LIN {X 0,Y 291.38,Z 152.183,A -85,B 0,C 180,E1 -16711.158,E2 -16711.158} C_VEL
LIN {X 0,Y 291.416,Z 152.178,A -85,B 0,C 180,E1 -16714.271,E2 -16714.271} C_VEL
LIN {X 0,Y 291.385,Z 152.183,A -85,B 0,C 180,E1 -16717.299,E2 -16717.299} C_VEL
LIN {X 0,Y 291.461,Z 152.175,A -85,B 0,C 180,E1 -16720.27,E2 -16720.27} C_VEL
LIN {X 0,Y 291.501,Z 152.17,A -85,B 0,C 180,E1 -16724.665,E2 -16724.665} C_VEL
LIN {X 0,Y 291.535,Z 152.322,A -85,B 0,C 180,E1 -16728.175,E2 -16728.175} C_VEL
LIN {X 0,Y 293.005,Z 156.516,A -85,B 0,C 180,E1 -16730.667,E2 -16730.667} C_VEL
LIN {X 0,Y 297.602,Z 162.945,A -85,B 0,C 180,E1 -16732.095,E2 -16732.095} C_VEL
LIN {X 0,Y 302.05,Z 169.865,A -85,B 0,C 180,E1 -16733.381,E2 -16733.381} C_VEL
LIN {X 0,Y 308.376,Z 180.311,A -85,B 0,C 180,E1 -16735.063,E2 -16735.063} C_VEL
LIN {X 0,Y 312.454,Z 188.42,A -85,B 0,C 180,E1 -16736.13,E2 -16736.13} C_VEL
LIN {X 0,Y 314.482,Z 193.12,A -85,B 0,C 180,E1 -16736.647,E2 -16736.647} C_VEL
LIN {X 0,Y 310.09,Z 262.242,A -85,B 0,C 180,E1 -16738.849,E2 -16738.849} C_VEL
LIN {X 0,Y 308.944,Z 275.275,A -85,B 0,C 180,E1 -16739.521,E2 -16739.521} C_VEL
LIN {X 0,Y 307.531,Z 287.536,A -85,B 0,C 180,E1 -16740.409,E2 -16740.409} C_VEL
LIN {X 0,Y 305.756,Z 299.005,A -85,B 0,C 180,E1 -16741.481,E2 -16741.481} C_VEL
LIN {X 0,Y 303.782,Z 309.929,A -85,B 0,C 180,E1 -16742.781,E2 -16742.781} C_VEL
LIN {X 0,Y 301.628,Z 320.38,A -85,B 0,C 180,E1 -16744.342,E2 -16744.342} C_VEL
LIN {X 0,Y 299.47,Z 329.569,A -85,B 0,C 180,E1 -16746.062,E2 -16746.062} C_VEL
LIN {X 0,Y 297.597,Z 336.876,A -85,B 0,C 180,E1 -16747.736,E2 -16747.736} C_VEL
LIN {X 0,Y 295.513,Z 344.591,A -85,B 0,C 180,E1 -16749.928,E2 -16749.928} C_VEL
LIN {X 0,Y 293.945,Z 350.077,A -85,B 0,C 180,E1 -16751.921,E2 -16751.921} C_VEL
LIN {X 0,Y 292.66,Z 354.329,A -85,B 0,C 180,E1 -16753.894,E2 -16753.894} C_VEL
LIN {X 0,Y 291.793,Z 357.055,A -85,B 0,C 180,E1 -16755.543,E2 -16755.543} C_VEL
LIN {X 0,Y 291.194,Z 358.762,A -85,B 0,C 180,E1 -16756.835,E2 -16756.835} C_VEL
LIN {X 0,Y 290.353,Z 360.927,A -85,B 0,C 180,E1 -16759.265,E2 -16759.265} C_VEL
LIN {X 0,Y 289.891,Z 361.74,A -85,B 0,C 180,E1 -16761.324,E2 -16761.324} C_VEL
LIN {X 0,Y 289.662,Z 361.742,A -85,B 0,C 180,E1 -16762.842,E2 -16762.842} C_VEL
LIN {X 0,Y 289.502,Z 361.254,A -85,B 0,C 180,E1 -16764.374,E2 -16764.374} C_VEL
LIN {X 0,Y 289.474,Z 360.131,A -85,B 0,C 180,E1 -16766.063,E2 -16766.063} C_VEL
LIN {X 0,Y 289.591,Z 357.737,A -85,B 0,C 180,E1 -16768.244,E2 -16768.244} C_VEL
LIN {X 0,Y 289.951,Z 353.898,A -85,B 0,C 180,E1 -16770.597,E2 -16770.597} C_VEL
LIN {X 0,Y 290.37,Z 348.539,A -85,B 0,C 180,E1 -16772.995,E2 -16772.995} C_VEL
LIN {X 0,Y 290.925,Z 342.639,A -85,B 0,C 180,E1 -16775.031,E2 -16775.031} C_VEL
LIN {X 0,Y 291.659,Z 335.36,A -85,B 0,C 180,E1 -16777.042,E2 -16777.042} C_VEL
LIN {X 0,Y 292.611,Z 326.228,A -85,B 0,C 180,E1 -16779.079,E2 -16779.079} C_VEL
LIN {X 0,Y 293.563,Z 317.163,A -85,B 0,C 180,E1 -16780.72,E2 -16780.72} C_VEL
LIN {X 0,Y 294.67,Z 306.188,A -85,B 0,C 180,E1 -16782.322,E2 -16782.322} C_VEL
LIN {X 0,Y 295.812,Z 293.704,A -85,B 0,C 180,E1 -16783.77,E2 -16783.77} C_VEL
LIN {X 0,Y 296.752,Z 280.809,A -85,B 0,C 180,E1 -16784.907,E2 -16784.907} C_VEL
LIN {X 0,Y 297.457,Z 267.609,A -85,B 0,C 180,E1 -16785.77,E2 -16785.77} C_VEL
LIN {X 0,Y 298.077,Z 253.321,A -85,B 0,C 180,E1 -16786.378,E2 -16786.378} C_VEL
LIN {X 0,Y 300.389,Z 178.97,A -85,B 0,C 180,E1 -16788.592,E2 -16788.592} C_VEL
LIN {X 0,Y 293.949,Z 159.621,A -85,B 0,C 180,E1 -16789.594,E2 -16789.594} C_VEL
LIN {X 0,Y 291.387,Z 152.189,A -85,B 0,C 180,E1 -16790.006,E2 -16790.006} C_VEL
LIN {X 0,Y 291.407,Z 152.184,A -85,B 0,C 180,E1 -16792.919,E2 -16792.919} C_VEL
LIN {X 0,Y 291.344,Z 152.192,A -85,B 0,C 180,E1 -16796.301,E2 -16796.301} C_VEL
LIN {X 0,Y 291.387,Z 152.187,A -85,B 0,C 180,E1 -16800.259,E2 -16800.259} C_VEL
LIN {X 0,Y 291.42,Z 152.182,A -85,B 0,C 180,E1 -16804.272,E2 -16804.272} C_VEL
LIN {X 0,Y 291.379,Z 152.192,A -85,B 0,C 180,E1 -16807.299,E2 -16807.299} C_VEL
LIN {X 0,Y 291.457,Z 152.177,A -85,B 0,C 180,E1 -16810.27,E2 -16810.27} C_VEL
LIN {X 0,Y 291.496,Z 152.173,A -85,B 0,C 180,E1 -16814.665,E2 -16814.665} C_VEL
LIN {X 0,Y 291.536,Z 152.171,A -85,B 0,C 180,E1 -16818.88,E2 -16818.88} C_VEL
LIN {X 0,Y 291.704,Z 152.147,A -85,B 0,C 180,E1 -16821.688,E2 -16821.688} C_VEL
LIN {X 0,Y 291.627,Z 152.157,A -85,B 0,C 180,E1 -16824.468,E2 -16824.468} C_VEL
LIN {X 0,Y 291.889,Z 152.127,A -85,B 0,C 180,E1 -16828.62,E2 -16828.62} C_VEL
LIN {X 0,Y 291.888,Z 152.124,A -85,B 0,C 180,E1 -16831.379,E2 -16831.379} C_VEL
LIN {X 0,Y 291.739,Z 152.145,A -85,B 0,C 180,E1 -16836.918,E2 -16836.918} C_VEL
LIN {X 0,Y 291.627,Z 152.156,A -85,B 0,C 180,E1 -16839.711,E2 -16839.711} C_VEL
LIN {X 0,Y 291.52,Z 152.17,A -85,B 0,C 180,E1 -16843.95,E2 -16843.95} C_VEL
LIN {X 0,Y 291.484,Z 152.176,A -85,B 0,C 180,E1 -16846.817,E2 -16846.817} C_VEL
LIN {X 0,Y 291.448,Z 152.179,A -85,B 0,C 180,E1 -16849.874,E2 -16849.874} C_VEL
LIN {X 0,Y 291.38,Z 152.191,A -85,B 0,C 180,E1 -16854.206,E2 -16854.206} C_VEL
LIN {X 0,Y 291.422,Z 152.181,A -85,B 0,C 180,E1 -16857.271,E2 -16857.271} C_VEL
LIN {X 0,Y 291.338,Z 152.195,A -85,B 0,C 180,E1 -16860.436,E2 -16860.436} C_VEL
LIN {X 0,Y 291.342,Z 152.193,A -85,B 0,C 180,E1 -16863.698,E2 -16863.698} C_VEL
LIN {X 0,Y 291.401,Z 152.184,A -85,B 0,C 180,E1 -16867.261,E2 -16867.261} C_VEL
LIN {X 0,Y 291.398,Z 152.185,A -85,B 0,C 180,E1 -16870.631,E2 -16870.631} C_VEL
LIN {X 0,Y 291.349,Z 152.191,A -85,B 0,C 180,E1 -16874.39,E2 -16874.39} C_VEL
LIN {X 0,Y 291.354,Z 152.191,A -85,B 0,C 180,E1 -16878.397,E2 -16878.397} C_VEL
LIN {X 0,Y 291.377,Z 152.188,A -85,B 0,C 180,E1 -16881.163,E2 -16881.163} C_VEL
LIN {X 0,Y 291.382,Z 152.186,A -85,B 0,C 180,E1 -16884.63,E2 -16884.63} C_VEL
LIN {X 0,Y 291.369,Z 152.19,A -85,B 0,C 180,E1 -16887.951,E2 -16887.951} C_VEL
LIN {X 0,Y 291.382,Z 152.188,A -85,B 0,C 180,E1 -16891.159,E2 -16891.159} C_VEL
LIN {X 0,Y 291.417,Z 152.182,A -85,B 0,C 180,E1 -16894.273,E2 -16894.273} C_VEL
LIN {X 0,Y 291.419,Z 152.182,A -85,B 0,C 180,E1 -16896.532,E2 -16896.532} C_VEL
LIN {X 0,Y 290.683,Z 152.277,A -85,B 0,C 180,E1 -16897.685,E2 -16897.685} C_VEL
LIN {X 0,Y 287.804,Z 152.634,A -85,B 0,C 180,E1 -16899.564,E2 -16899.564} C_VEL
LIN {X 0,Y 285.435,Z 152.93,A -85,B 0,C 180,E1 -16901.089,E2 -16901.089} C_VEL
LIN {X 0,Y 284.47,Z 153.047,A -85,B 0,C 180,E1 -16902.271,E2 -16902.271} C_VEL
LIN {X 0,Y 284.417,Z 153.055,A -85,B 0,C 180,E1 -16902.67,E2 -16902.67} C_VEL
LIN {X 0,Y 284.479,Z 153.047,A -85,B 0,C 180,E1 -16905.698,E2 -16905.698} C_VEL
LIN {X 0,Y 284.564,Z 153.036,A -85,B 0,C 180,E1 -16910.045,E2 -16910.045} C_VEL
LIN {X 0,Y 284.691,Z 153.024,A -85,B 0,C 180,E1 -16912.91,E2 -16912.91} C_VEL
LIN {X 0,Y 284.854,Z 153.002,A -85,B 0,C 180,E1 -16918.587,E2 -16918.587} C_VEL
LIN {X 0,Y 284.854,Z 153,A -85,B 0,C 180,E1 -16921.414,E2 -16921.414} C_VEL
LIN {X 0,Y 284.697,Z 153.021,A -85,B 0,C 180,E1 -16927.091,E2 -16927.091} C_VEL
LIN {X 0,Y 284.565,Z 153.036,A -85,B 0,C 180,E1 -16929.956,E2 -16929.956} C_VEL
LIN {X 0,Y 284.48,Z 153.048,A -85,B 0,C 180,E1 -16934.303,E2 -16934.303} C_VEL
LIN {X 0,Y 284.424,Z 153.053,A -85,B 0,C 180,E1 -16937.249,E2 -16937.249} C_VEL
LIN {X 0,Y 284.376,Z 153.062,A -85,B 0,C 180,E1 -16940.243,E2 -16940.243} C_VEL
LIN {X 0,Y 284.338,Z 153.065,A -85,B 0,C 180,E1 -16944.847,E2 -16944.847} C_VEL
LIN {X 0,Y 284.331,Z 153.067,A -85,B 0,C 180,E1 -16948.011,E2 -16948.011} C_VEL
LIN {X 0,Y 284.295,Z 153.069,A -85,B 0,C 180,E1 -16951.275,E2 -16951.275} C_VEL
LIN {X 0,Y 284.362,Z 153.061,A -85,B 0,C 180,E1 -16955.355,E2 -16955.355} C_VEL
LIN {X 0,Y 284.334,Z 153.068,A -85,B 0,C 180,E1 -16958.166,E2 -16958.166} C_VEL
LIN {X 0,Y 284.302,Z 153.073,A -85,B 0,C 180,E1 -16961.871,E2 -16961.871} C_VEL
LIN {X 0,Y 284.256,Z 153.077,A -85,B 0,C 180,E1 -16966.19,E2 -16966.19} C_VEL
LIN {X 0,Y 284.307,Z 153.071,A -85,B 0,C 180,E1 -16970.025,E2 -16970.025} C_VEL
LIN {X 0,Y 284.335,Z 153.07,A -85,B 0,C 180,E1 -16973.615,E2 -16973.615} C_VEL
LIN {X 0,Y 284.385,Z 153.189,A -85,B 0,C 180,E1 -16976.591,E2 -16976.591} C_VEL
LIN {X 0,Y 287.211,Z 166.814,A -85,B 0,C 180,E1 -16980.7,E2 -16980.7} C_VEL
LIN {X 0,Y 288.505,Z 174.149,A -85,B 0,C 180,E1 -16982.823,E2 -16982.823} C_VEL
LIN {X 0,Y 287.7,Z 181.099,A -85,B 0,C 180,E1 -16984.669,E2 -16984.669} C_VEL
LIN {X 0,Y 292.734,Z 226.959,A -85,B 0,C 180,E1 -16986.473,E2 -16986.473} C_VEL
LIN {X 0,Y 290.738,Z 290.445,A -85,B 0,C 180,E1 -16988.462,E2 -16988.462} C_VEL
LIN {X 0,Y 289.869,Z 303.747,A -85,B 0,C 180,E1 -16989.139,E2 -16989.139} C_VEL
LIN {X 0,Y 288.82,Z 316.65,A -85,B 0,C 180,E1 -16990.083,E2 -16990.083} C_VEL
LIN {X 0,Y 287.576,Z 328.945,A -85,B 0,C 180,E1 -16991.292,E2 -16991.292} C_VEL
LIN {X 0,Y 286.423,Z 340.122,A -85,B 0,C 180,E1 -16992.692,E2 -16992.692} C_VEL
LIN {X 0,Y 285.103,Z 351.202,A -85,B 0,C 180,E1 -16994.451,E2 -16994.451} C_VEL
LIN {X 0,Y 284.188,Z 361.095,A -85,B 0,C 180,E1 -16996.413,E2 -16996.413} C_VEL
LIN {X 0,Y 283.318,Z 369.657,A -85,B 0,C 180,E1 -16998.554,E2 -16998.554} C_VEL
LIN {X 0,Y 282.878,Z 376.54,A -85,B 0,C 180,E1 -17000.707,E2 -17000.707} C_VEL
LIN {X 0,Y 282.641,Z 381.978,A -85,B 0,C 180,E1 -17002.859,E2 -17002.859} C_VEL
LIN {X 0,Y 282.629,Z 386.148,A -85,B 0,C 180,E1 -17005.008,E2 -17005.008} C_VEL
LIN {X 0,Y 282.569,Z 389.15,A -85,B 0,C 180,E1 -17007.149,E2 -17007.149} C_VEL
LIN {X 0,Y 282.65,Z 390.559,A -85,B 0,C 180,E1 -17008.576,E2 -17008.576} C_VEL
LIN {X 0,Y 282.778,Z 391.518,A -85,B 0,C 180,E1 -17010.001,E2 -17010.001} C_VEL
LIN {X 0,Y 282.516,Z 392.026,A -85,B 0,C 180,E1 -17011.426,E2 -17011.426} C_VEL
LIN {X 0,Y 282.467,Z 392.128,A -85,B 0,C 180,E1 -17012.853,E2 -17012.853} C_VEL
LIN {X 0,Y 282.361,Z 391.221,A -85,B 0,C 180,E1 -17015.369,E2 -17015.369} C_VEL
LIN {X 0,Y 282.481,Z 389.817,A -85,B 0,C 180,E1 -17017.146,E2 -17017.146} C_VEL
LIN {X 0,Y 282.883,Z 387.242,A -85,B 0,C 180,E1 -17019.294,E2 -17019.294} C_VEL
LIN {X 0,Y 283.555,Z 383.662,A -85,B 0,C 180,E1 -17021.437,E2 -17021.437} C_VEL
LIN {X 0,Y 284.651,Z 378.997,A -85,B 0,C 180,E1 -17023.566,E2 -17023.566} C_VEL
LIN {X 0,Y 286.499,Z 372.036,A -85,B 0,C 180,E1 -17026.02,E2 -17026.02} C_VEL
LIN {X 0,Y 288.067,Z 365.342,A -85,B 0,C 180,E1 -17027.918,E2 -17027.918} C_VEL
LIN {X 0,Y 290.261,Z 357.026,A -85,B 0,C 180,E1 -17029.815,E2 -17029.815} C_VEL
LIN {X 0,Y 292.489,Z 347.996,A -85,B 0,C 180,E1 -17031.496,E2 -17031.496} C_VEL
LIN {X 0,Y 295.2,Z 336.973,A -85,B 0,C 180,E1 -17033.131,E2 -17033.131} C_VEL
LIN {X 0,Y 297.777,Z 324.554,A -85,B 0,C 180,E1 -17034.581,E2 -17034.581} C_VEL
LIN {X 0,Y 300.056,Z 312.388,A -85,B 0,C 180,E1 -17035.678,E2 -17035.678} C_VEL
LIN {X 0,Y 302.163,Z 298.433,A -85,B 0,C 180,E1 -17036.599,E2 -17036.599} C_VEL
LIN {X 0,Y 303.623,Z 285.304,A -85,B 0,C 180,E1 -17037.204,E2 -17037.204} C_VEL
LIN {X 0,Y 307.025,Z 230.877,A -85,B 0,C 180,E1 -17038.964,E2 -17038.964} C_VEL
LIN {X 0,Y 305.371,Z 215.387,A -85,B 0,C 180,E1 -17039.917,E2 -17039.917} C_VEL
LIN {X 0,Y 303.242,Z 201.67,A -85,B 0,C 180,E1 -17040.919,E2 -17040.919} C_VEL
LIN {X 0,Y 301.932,Z 196.07,A -85,B 0,C 180,E1 -17041.414,E2 -17041.414} C_VEL
LIN {X 0,Y 298.299,Z 188.202,A -85,B 0,C 180,E1 -17042.513,E2 -17042.513} C_VEL
LIN {X 0,Y 295.654,Z 183.064,A -85,B 0,C 180,E1 -17043.325,E2 -17043.325} C_VEL
LIN {X 0,Y 293.062,Z 178.27,A -85,B 0,C 180,E1 -17044.153,E2 -17044.153} C_VEL
LIN {X 0,Y 290.719,Z 173.805,A -85,B 0,C 180,E1 -17044.99,E2 -17044.99} C_VEL
LIN {X 0,Y 288.987,Z 167.269,A -85,B 0,C 180,E1 -17047.89,E2 -17047.89} C_VEL
LIN {X 0,Y 287.252,Z 161.816,A -85,B 0,C 180,E1 -17050.671,E2 -17050.671} C_VEL
LIN {X 0,Y 285.585,Z 156.926,A -85,B 0,C 180,E1 -17053.556,E2 -17053.556} C_VEL
LIN {X 0,Y 284.264,Z 153.07,A -85,B 0,C 180,E1 -17056.304,E2 -17056.304} C_VEL
LIN {X 0,Y 284.311,Z 153.065,A -85,B 0,C 180,E1 -17060.024,E2 -17060.024} C_VEL
LIN {X 0,Y 284.346,Z 153.055,A -85,B 0,C 180,E1 -17063.615,E2 -17063.615} C_VEL
LIN {X 0,Y 284.311,Z 153.067,A -85,B 0,C 180,E1 -17067.19,E2 -17067.19} C_VEL
LIN {X 0,Y 284.359,Z 153.063,A -85,B 0,C 180,E1 -17070.375,E2 -17070.375} C_VEL
LIN {X 0,Y 284.378,Z 153.057,A -85,B 0,C 180,E1 -17073.586,E2 -17073.586} C_VEL
LIN {X 0,Y 284.37,Z 153.056,A -85,B 0,C 180,E1 -17076.707,E2 -17076.707} C_VEL
LIN {X 0,Y 284.39,Z 153.057,A -85,B 0,C 180,E1 -17081.26,E2 -17081.26} C_VEL
LIN {X 0,Y 284.486,Z 153.078,A -85,B 0,C 180,E1 -17085.925,E2 -17085.925} C_VEL
LIN {X 0,Y 285.838,Z 157.286,A -85,B 0,C 180,E1 -17088.833,E2 -17088.833} C_VEL
LIN {X 0,Y 289.338,Z 161.911,A -85,B 0,C 180,E1 -17090.064,E2 -17090.064} C_VEL
LIN {X 0,Y 294.079,Z 168.576,A -85,B 0,C 180,E1 -17091.598,E2 -17091.598} C_VEL
LIN {X 0,Y 298.738,Z 176.141,A -85,B 0,C 180,E1 -17093.011,E2 -17093.011} C_VEL
LIN {X 0,Y 304.057,Z 185.069,A -85,B 0,C 180,E1 -17094.499,E2 -17094.499} C_VEL
LIN {X 0,Y 308.04,Z 193.204,A -85,B 0,C 180,E1 -17095.583,E2 -17095.583} C_VEL
LIN {X 0,Y 308.957,Z 195.331,A -85,B 0,C 180,E1 -17095.838,E2 -17095.838} C_VEL
LIN {X 0,Y 304.461,Z 262.962,A -85,B 0,C 180,E1 -17098.057,E2 -17098.057} C_VEL
LIN {X 0,Y 303.369,Z 274.844,A -85,B 0,C 180,E1 -17098.672,E2 -17098.672} C_VEL
LIN {X 0,Y 301.849,Z 287.601,A -85,B 0,C 180,E1 -17099.597,E2 -17099.597} C_VEL
LIN {X 0,Y 299.973,Z 298.978,A -85,B 0,C 180,E1 -17100.671,E2 -17100.671} C_VEL
LIN {X 0,Y 297.818,Z 310.192,A -85,B 0,C 180,E1 -17102.028,E2 -17102.028} C_VEL
LIN {X 0,Y 295.496,Z 320.768,A -85,B 0,C 180,E1 -17103.631,E2 -17103.631} C_VEL
LIN {X 0,Y 293.053,Z 330.567,A -85,B 0,C 180,E1 -17105.504,E2 -17105.504} C_VEL
LIN {X 0,Y 290.692,Z 339.209,A -85,B 0,C 180,E1 -17107.582,E2 -17107.582} C_VEL
LIN {X 0,Y 288.54,Z 346.426,A -85,B 0,C 180,E1 -17109.816,E2 -17109.816} C_VEL
LIN {X 0,Y 286.724,Z 352.17,A -85,B 0,C 180,E1 -17112.114,E2 -17112.114} C_VEL
LIN {X 0,Y 285.386,Z 356.243,A -85,B 0,C 180,E1 -17114.256,E2 -17114.256} C_VEL
LIN {X 0,Y 284.603,Z 358.427,A -85,B 0,C 180,E1 -17115.761,E2 -17115.761} C_VEL
LIN {X 0,Y 283.959,Z 360.095,A -85,B 0,C 180,E1 -17117.277,E2 -17117.277} C_VEL
LIN {X 0,Y 283.241,Z 361.645,A -85,B 0,C 180,E1 -17119.457,E2 -17119.457} C_VEL
LIN {X 0,Y 282.716,Z 362.222,A -85,B 0,C 180,E1 -17121.893,E2 -17121.893} C_VEL
LIN {X 0,Y 282.509,Z 361.969,A -85,B 0,C 180,E1 -17123.455,E2 -17123.455} C_VEL
LIN {X 0,Y 282.377,Z 361.171,A -85,B 0,C 180,E1 -17125.03,E2 -17125.03} C_VEL
LIN {X 0,Y 282.383,Z 359.89,A -85,B 0,C 180,E1 -17126.614,E2 -17126.614} C_VEL
LIN {X 0,Y 282.487,Z 358.017,A -85,B 0,C 180,E1 -17128.209,E2 -17128.209} C_VEL
LIN {X 0,Y 282.852,Z 354.119,A -85,B 0,C 180,E1 -17130.621,E2 -17130.621} C_VEL
LIN {X 0,Y 283.3,Z 348.691,A -85,B 0,C 180,E1 -17133.076,E2 -17133.076} C_VEL
LIN {X 0,Y 283.892,Z 342.518,A -85,B 0,C 180,E1 -17135.219,E2 -17135.219} C_VEL
LIN {X 0,Y 284.778,Z 334.003,A -85,B 0,C 180,E1 -17137.559,E2 -17137.559} C_VEL
LIN {X 0,Y 285.74,Z 325.021,A -85,B 0,C 180,E1 -17139.524,E2 -17139.524} C_VEL
LIN {X 0,Y 286.866,Z 314.271,A -85,B 0,C 180,E1 -17141.412,E2 -17141.412} C_VEL
LIN {X 0,Y 287.995,Z 303.415,A -85,B 0,C 180,E1 -17142.937,E2 -17142.937} C_VEL
LIN {X 0,Y 289.063,Z 290.684,A -85,B 0,C 180,E1 -17144.346,E2 -17144.346} C_VEL
LIN {X 0,Y 289.963,Z 279.04,A -85,B 0,C 180,E1 -17145.34,E2 -17145.34} C_VEL
LIN {X 0,Y 290.673,Z 265.528,A -85,B 0,C 180,E1 -17146.185,E2 -17146.185} C_VEL
LIN {X 0,Y 291.272,Z 251.705,A -85,B 0,C 180,E1 -17146.75,E2 -17146.75} C_VEL
LIN {X 0,Y 293.552,Z 180.316,A -85,B 0,C 180,E1 -17148.943,E2 -17148.943} C_VEL
LIN {X 0,Y 287.659,Z 162.583,A -85,B 0,C 180,E1 -17149.88,E2 -17149.88} C_VEL
LIN {X 0,Y 284.357,Z 153.063,A -85,B 0,C 180,E1 -17150.431,E2 -17150.431} C_VEL
LIN {X 0,Y 284.34,Z 153.064,A -85,B 0,C 180,E1 -17154.651,E2 -17154.651} C_VEL
LIN {X 0,Y 284.295,Z 153.07,A -85,B 0,C 180,E1 -17158.725,E2 -17158.725} C_VEL
LIN {X 0,Y 284.399,Z 153.059,A -85,B 0,C 180,E1 -17162.825,E2 -17162.825} C_VEL
LIN {X 0,Y 284.365,Z 153.062,A -85,B 0,C 180,E1 -17166.706,E2 -17166.706} C_VEL
LIN {X 0,Y 284.368,Z 153.065,A -85,B 0,C 180,E1 -17171.259,E2 -17171.259} C_VEL
LIN {X 0,Y 284.462,Z 153.048,A -85,B 0,C 180,E1 -17175.696,E2 -17175.696} C_VEL
LIN {X 0,Y 284.565,Z 153.036,A -85,B 0,C 180,E1 -17180.044,E2 -17180.044} C_VEL
LIN {X 0,Y 284.692,Z 153.024,A -85,B 0,C 180,E1 -17182.909,E2 -17182.909} C_VEL
LIN {X 0,Y 284.854,Z 153.002,A -85,B 0,C 180,E1 -17188.586,E2 -17188.586} C_VEL
LIN {X 0,Y 284.854,Z 153,A -85,B 0,C 180,E1 -17191.413,E2 -17191.413} C_VEL
LIN {X 0,Y 284.692,Z 153.022,A -85,B 0,C 180,E1 -17197.09,E2 -17197.09} C_VEL
LIN {X 0,Y 284.564,Z 153.036,A -85,B 0,C 180,E1 -17199.955,E2 -17199.955} C_VEL
LIN {X 0,Y 284.479,Z 153.049,A -85,B 0,C 180,E1 -17204.302,E2 -17204.302} C_VEL
LIN {X 0,Y 284.423,Z 153.053,A -85,B 0,C 180,E1 -17207.248,E2 -17207.248} C_VEL
LIN {X 0,Y 284.375,Z 153.062,A -85,B 0,C 180,E1 -17210.242,E2 -17210.242} C_VEL
LIN {X 0,Y 284.336,Z 153.065,A -85,B 0,C 180,E1 -17214.846,E2 -17214.846} C_VEL
LIN {X 0,Y 284.361,Z 153.063,A -85,B 0,C 180,E1 -17218.007,E2 -17218.007} C_VEL
LIN {X 0,Y 284.296,Z 153.069,A -85,B 0,C 180,E1 -17221.274,E2 -17221.274} C_VEL
LIN {X 0,Y 284.359,Z 153.061,A -85,B 0,C 180,E1 -17225.354,E2 -17225.354} C_VEL
LIN {X 0,Y 284.332,Z 153.068,A -85,B 0,C 180,E1 -17228.165,E2 -17228.165} C_VEL
LIN {X 0,Y 284.338,Z 153.066,A -85,B 0,C 180,E1 -17232.14,E2 -17232.14} C_VEL
LIN {X 0,Y 284.315,Z 153.069,A -85,B 0,C 180,E1 -17236.201,E2 -17236.201} C_VEL
LIN {X 0,Y 284.348,Z 153.065,A -85,B 0,C 180,E1 -17240.013,E2 -17240.013} C_VEL
LIN {X 0,Y 284.349,Z 153.066,A -85,B 0,C 180,E1 -17243.617,E2 -17243.617} C_VEL
LIN {X 0,Y 284.305,Z 153.07,A -85,B 0,C 180,E1 -17247.19,E2 -17247.19} C_VEL
LIN {X 0,Y 284.356,Z 153.061,A -85,B 0,C 180,E1 -17250.376,E2 -17250.376} C_VEL
LIN {X 0,Y 284.377,Z 153.063,A -85,B 0,C 180,E1 -17253.587,E2 -17253.587} C_VEL
LIN {X 0,Y 284.363,Z 153.061,A -85,B 0,C 180,E1 -17256.707,E2 -17256.707} C_VEL
LIN {X 0,Y 284.401,Z 153.06,A -85,B 0,C 180,E1 -17261.262,E2 -17261.262} C_VEL
LIN {X 0,Y 284.417,Z 153.055,A -85,B 0,C 180,E1 -17262.67,E2 -17262.67} C_VEL
LIN {X 0,Y 283.809,Z 153.135,A -85,B 0,C 180,E1 -17263.853,E2 -17263.853} C_VEL
LIN {X 0,Y 280.963,Z 153.489,A -85,B 0,C 180,E1 -17265.779,E2 -17265.779} C_VEL
LIN {X 0,Y 278.528,Z 153.79,A -85,B 0,C 180,E1 -17267.344,E2 -17267.344} C_VEL
LIN {X 0,Y 277.509,Z 153.915,A -85,B 0,C 180,E1 -17268.558,E2 -17268.558} C_VEL
LIN {X 0,Y 277.442,Z 153.92,A -85,B 0,C 180,E1 -17268.969,E2 -17268.969} C_VEL
LIN {X 0,Y 277.611,Z 153.905,A -85,B 0,C 180,E1 -17271.264,E2 -17271.264} C_VEL
LIN {X 0,Y 277.567,Z 153.907,A -85,B 0,C 180,E1 -17274.188,E2 -17274.188} C_VEL
LIN {X 0,Y 277.82,Z 153.878,A -85,B 0,C 180,E1 -17278.551,E2 -17278.551} C_VEL
LIN {X 0,Y 277.82,Z 153.876,A -85,B 0,C 180,E1 -17281.45,E2 -17281.45} C_VEL
LIN {X 0,Y 277.652,Z 153.898,A -85,B 0,C 180,E1 -17287.271,E2 -17287.271} C_VEL
LIN {X 0,Y 277.505,Z 153.917,A -85,B 0,C 180,E1 -17290.212,E2 -17290.212} C_VEL
LIN {X 0,Y 277.433,Z 153.928,A -85,B 0,C 180,E1 -17294.675,E2 -17294.675} C_VEL
LIN {X 0,Y 277.344,Z 153.935,A -85,B 0,C 180,E1 -17299.234,E2 -17299.234} C_VEL
LIN {X 0,Y 277.291,Z 153.945,A -85,B 0,C 180,E1 -17304.159,E2 -17304.159} C_VEL
LIN {X 0,Y 277.325,Z 153.937,A -85,B 0,C 180,E1 -17307.506,E2 -17307.506} C_VEL
LIN {X 0,Y 277.271,Z 153.947,A -85,B 0,C 180,E1 -17310.482,E2 -17310.482} C_VEL
LIN {X 0,Y 277.254,Z 153.949,A -85,B 0,C 180,E1 -17313.895,E2 -17313.895} C_VEL
LIN {X 0,Y 277.289,Z 153.941,A -85,B 0,C 180,E1 -17317.467,E2 -17317.467} C_VEL
LIN {X 0,Y 277.24,Z 153.949,A -85,B 0,C 180,E1 -17321.232,E2 -17321.232} C_VEL
LIN {X 0,Y 277.204,Z 153.952,A -85,B 0,C 180,E1 -17325.227,E2 -17325.227} C_VEL
LIN {X 0,Y 277.223,Z 153.953,A -85,B 0,C 180,E1 -17329.513,E2 -17329.513} C_VEL
LIN {X 0,Y 277.272,Z 153.946,A -85,B 0,C 180,E1 -17332.532,E2 -17332.532} C_VEL
LIN {X 0,Y 277.381,Z 154.102,A -85,B 0,C 180,E1 -17336.305,E2 -17336.305} C_VEL
LIN {X 0,Y 280.232,Z 168.104,A -85,B 0,C 180,E1 -17340.629,E2 -17340.629} C_VEL
LIN {X 0,Y 281.433,Z 174.352,A -85,B 0,C 180,E1 -17342.485,E2 -17342.485} C_VEL
LIN {X 0,Y 280.788,Z 180.51,A -85,B 0,C 180,E1 -17344.196,E2 -17344.196} C_VEL
LIN {X 0,Y 285.793,Z 228.759,A -85,B 0,C 180,E1 -17346.17,E2 -17346.17} C_VEL
LIN {X 0,Y 283.741,Z 290.888,A -85,B 0,C 180,E1 -17348.19,E2 -17348.19} C_VEL
LIN {X 0,Y 282.888,Z 303.945,A -85,B 0,C 180,E1 -17348.886,E2 -17348.886} C_VEL
LIN {X 0,Y 281.914,Z 315.678,A -85,B 0,C 180,E1 -17349.764,E2 -17349.764} C_VEL
LIN {X 0,Y 280.842,Z 326.533,A -85,B 0,C 180,E1 -17350.826,E2 -17350.826} C_VEL
LIN {X 0,Y 279.591,Z 338.05,A -85,B 0,C 180,E1 -17352.256,E2 -17352.256} C_VEL
LIN {X 0,Y 278.329,Z 348.506,A -85,B 0,C 180,E1 -17353.874,E2 -17353.874} C_VEL
LIN {X 0,Y 277.374,Z 357.955,A -85,B 0,C 180,E1 -17355.698,E2 -17355.698} C_VEL
LIN {X 0,Y 276.479,Z 367.122,A -85,B 0,C 180,E1 -17357.895,E2 -17357.895} C_VEL
LIN {X 0,Y 275.889,Z 374.443,A -85,B 0,C 180,E1 -17360.099,E2 -17360.099} C_VEL
LIN {X 0,Y 275.664,Z 379.38,A -85,B 0,C 180,E1 -17361.94,E2 -17361.94} C_VEL
LIN {X 0,Y 275.573,Z 384.9,A -85,B 0,C 180,E1 -17364.617,E2 -17364.617} C_VEL
LIN {X 0,Y 275.497,Z 388.467,A -85,B 0,C 180,E1 -17367.076,E2 -17367.076} C_VEL
LIN {X 0,Y 275.562,Z 389.974,A -85,B 0,C 180,E1 -17368.539,E2 -17368.539} C_VEL
LIN {X 0,Y 275.707,Z 390.989,A -85,B 0,C 180,E1 -17370.001,E2 -17370.001} C_VEL
LIN {X 0,Y 275.431,Z 391.544,A -85,B 0,C 180,E1 -17371.463,E2 -17371.463} C_VEL
LIN {X 0,Y 275.389,Z 391.701,A -85,B 0,C 180,E1 -17372.926,E2 -17372.926} C_VEL
LIN {X 0,Y 275.274,Z 391.033,A -85,B 0,C 180,E1 -17375.305,E2 -17375.305} C_VEL
LIN {X 0,Y 275.416,Z 389.592,A -85,B 0,C 180,E1 -17377.331,E2 -17377.331} C_VEL
LIN {X 0,Y 275.678,Z 388.066,A -85,B 0,C 180,E1 -17378.799,E2 -17378.799} C_VEL
LIN {X 0,Y 276.291,Z 384.93,A -85,B 0,C 180,E1 -17380.999,E2 -17380.999} C_VEL
LIN {X 0,Y 277.253,Z 380.767,A -85,B 0,C 180,E1 -17383.188,E2 -17383.188} C_VEL
LIN {X 0,Y 279.097,Z 374.492,A -85,B 0,C 180,E1 -17385.706,E2 -17385.706} C_VEL
LIN {X 0,Y 280.658,Z 368.195,A -85,B 0,C 180,E1 -17387.714,E2 -17387.714} C_VEL
LIN {X 0,Y 283.166,Z 359.297,A -85,B 0,C 180,E1 -17389.955,E2 -17389.955} C_VEL
LIN {X 0,Y 285.544,Z 350.822,A -85,B 0,C 180,E1 -17391.666,E2 -17391.666} C_VEL
LIN {X 0,Y 288.182,Z 340.642,A -85,B 0,C 180,E1 -17393.347,E2 -17393.347} C_VEL
LIN {X 0,Y 290.832,Z 329.342,A -85,B 0,C 180,E1 -17394.827,E2 -17394.827} C_VEL
LIN {X 0,Y 293.062,Z 318.51,A -85,B 0,C 180,E1 -17395.955,E2 -17395.955} C_VEL
LIN {X 0,Y 295.428,Z 305.654,A -85,B 0,C 180,E1 -17396.968,E2 -17396.968} C_VEL
LIN {X 0,Y 297.324,Z 292.234,A -85,B 0,C 180,E1 -17397.734,E2 -17397.734} C_VEL
LIN {X 0,Y 298.511,Z 278.399,A -85,B 0,C 180,E1 -17398.286,E2 -17398.286} C_VEL
LIN {X 0,Y 301.63,Z 231.913,A -85,B 0,C 180,E1 -17399.823,E2 -17399.823} C_VEL
LIN {X 0,Y 300.144,Z 217.266,A -85,B 0,C 180,E1 -17400.756,E2 -17400.756} C_VEL
LIN {X 0,Y 298.09,Z 203.527,A -85,B 0,C 180,E1 -17401.801,E2 -17401.801} C_VEL
LIN {X 0,Y 297.145,Z 199.472,A -85,B 0,C 180,E1 -17402.191,E2 -17402.191} C_VEL
LIN {X 0,Y 292.378,Z 189.282,A -85,B 0,C 180,E1 -17403.715,E2 -17403.715} C_VEL
LIN {X 0,Y 289.167,Z 183.227,A -85,B 0,C 180,E1 -17404.805,E2 -17404.805} C_VEL
LIN {X 0,Y 286.288,Z 178.143,A -85,B 0,C 180,E1 -17405.811,E2 -17405.811} C_VEL
LIN {X 0,Y 283.402,Z 172.87,A -85,B 0,C 180,E1 -17406.974,E2 -17406.974} C_VEL
LIN {X 0,Y 281.353,Z 165.939,A -85,B 0,C 180,E1 -17410.502,E2 -17410.502} C_VEL
LIN {X 0,Y 279.844,Z 161.324,A -85,B 0,C 180,E1 -17413.255,E2 -17413.255} C_VEL
LIN {X 0,Y 277.962,Z 156.287,A -85,B 0,C 180,E1 -17416.947,E2 -17416.947} C_VEL
LIN {X 0,Y 277.219,Z 153.946,A -85,B 0,C 180,E1 -17418.981,E2 -17418.981} C_VEL
LIN {X 0,Y 277.278,Z 153.939,A -85,B 0,C 180,E1 -17422.532,E2 -17422.532} C_VEL
LIN {X 0,Y 277.25,Z 153.939,A -85,B 0,C 180,E1 -17426.104,E2 -17426.104} C_VEL
LIN {X 0,Y 277.265,Z 153.942,A -85,B 0,C 180,E1 -17429.538,E2 -17429.538} C_VEL
LIN {X 0,Y 277.359,Z 153.938,A -85,B 0,C 180,E1 -17432.864,E2 -17432.864} C_VEL
LIN {X 0,Y 277.332,Z 153.937,A -85,B 0,C 180,E1 -17436.079,E2 -17436.079} C_VEL
LIN {X 0,Y 277.339,Z 153.939,A -85,B 0,C 180,E1 -17440.765,E2 -17440.765} C_VEL
LIN {X 0,Y 277.38,Z 154.051,A -85,B 0,C 180,E1 -17443.249,E2 -17443.249} C_VEL
LIN {X 0,Y 278.922,Z 158.39,A -85,B 0,C 180,E1 -17446.8,E2 -17446.8} C_VEL
LIN {X 0,Y 283.76,Z 164.76,A -85,B 0,C 180,E1 -17448.718,E2 -17448.718} C_VEL
LIN {X 0,Y 287.805,Z 170.198,A -85,B 0,C 180,E1 -17450.157,E2 -17450.157} C_VEL
LIN {X 0,Y 291.822,Z 176.006,A -85,B 0,C 180,E1 -17451.474,E2 -17451.474} C_VEL
LIN {X 0,Y 299.937,Z 190.072,A -85,B 0,C 180,E1 -17453.95,E2 -17453.95} C_VEL
LIN {X 0,Y 303.511,Z 197.695,A -85,B 0,C 180,E1 -17454.983,E2 -17454.983} C_VEL
LIN {X 0,Y 303.526,Z 199.582,A -85,B 0,C 180,E1 -17455.073,E2 -17455.073} C_VEL
LIN {X 0,Y 298.932,Z 263.581,A -85,B 0,C 180,E1 -17457.22,E2 -17457.22} C_VEL
LIN {X 0,Y 297.719,Z 275.916,A -85,B 0,C 180,E1 -17457.886,E2 -17457.886} C_VEL
LIN {X 0,Y 296.15,Z 288.185,A -85,B 0,C 180,E1 -17458.795,E2 -17458.795} C_VEL
LIN {X 0,Y 293.976,Z 300.594,A -85,B 0,C 180,E1 -17459.999,E2 -17459.999} C_VEL
LIN {X 0,Y 291.732,Z 311.621,A -85,B 0,C 180,E1 -17461.38,E2 -17461.38} C_VEL
LIN {X 0,Y 289.585,Z 320.674,A -85,B 0,C 180,E1 -17462.782,E2 -17462.782} C_VEL
LIN {X 0,Y 287.173,Z 329.927,A -85,B 0,C 180,E1 -17464.561,E2 -17464.561} C_VEL
LIN {X 0,Y 284.527,Z 338.987,A -85,B 0,C 180,E1 -17466.737,E2 -17466.737} C_VEL
LIN {X 0,Y 282.28,Z 346.198,A -85,B 0,C 180,E1 -17468.952,E2 -17468.952} C_VEL
LIN {X 0,Y 280.631,Z 351.062,A -85,B 0,C 180,E1 -17470.825,E2 -17470.825} C_VEL
LIN {X 0,Y 278.996,Z 355.636,A -85,B 0,C 180,E1 -17473.103,E2 -17473.103} C_VEL
LIN {X 0,Y 277.523,Z 359.44,A -85,B 0,C 180,E1 -17475.779,E2 -17475.779} C_VEL
LIN {X 0,Y 276.719,Z 361.277,A -85,B 0,C 180,E1 -17477.744,E2 -17477.744} C_VEL
LIN {X 0,Y 276.12,Z 362.342,A -85,B 0,C 180,E1 -17479.651,E2 -17479.651} C_VEL
LIN {X 0,Y 275.813,Z 362.633,A -85,B 0,C 180,E1 -17480.899,E2 -17480.899} C_VEL
LIN {X 0,Y 275.429,Z 362.353,A -85,B 0,C 180,E1 -17483.277,E2 -17483.277} C_VEL
LIN {X 0,Y 275.271,Z 360.912,A -85,B 0,C 180,E1 -17485.723,E2 -17485.723} C_VEL
LIN {X 0,Y 275.392,Z 358.277,A -85,B 0,C 180,E1 -17488.171,E2 -17488.171} C_VEL
LIN {X 0,Y 275.763,Z 354.332,A -85,B 0,C 180,E1 -17490.644,E2 -17490.644} C_VEL
LIN {X 0,Y 276.156,Z 349.532,A -85,B 0,C 180,E1 -17492.877,E2 -17492.877} C_VEL
LIN {X 0,Y 276.811,Z 342.829,A -85,B 0,C 180,E1 -17495.281,E2 -17495.281} C_VEL
LIN {X 0,Y 277.578,Z 335.304,A -85,B 0,C 180,E1 -17497.42,E2 -17497.42} C_VEL
LIN {X 0,Y 278.641,Z 325.952,A -85,B 0,C 180,E1 -17499.558,E2 -17499.558} C_VEL
LIN {X 0,Y 279.623,Z 316.509,A -85,B 0,C 180,E1 -17501.295,E2 -17501.295} C_VEL
LIN {X 0,Y 280.804,Z 305.57,A -85,B 0,C 180,E1 -17502.926,E2 -17502.926} C_VEL
LIN {X 0,Y 281.877,Z 294.262,A -85,B 0,C 180,E1 -17504.276,E2 -17504.276} C_VEL
LIN {X 0,Y 282.879,Z 281.456,A -85,B 0,C 180,E1 -17505.457,E2 -17505.457} C_VEL
LIN {X 0,Y 283.595,Z 268.334,A -85,B 0,C 180,E1 -17506.359,E2 -17506.359} C_VEL
LIN {X 0,Y 284.256,Z 254.641,A -85,B 0,C 180,E1 -17506.978,E2 -17506.978} C_VEL
LIN {X 0,Y 286.709,Z 181.629,A -85,B 0,C 180,E1 -17509.294,E2 -17509.294} C_VEL
LIN {X 0,Y 281.208,Z 165.086,A -85,B 0,C 180,E1 -17510.196,E2 -17510.196} C_VEL
LIN {X 0,Y 277.302,Z 153.942,A -85,B 0,C 180,E1 -17510.877,E2 -17510.877} C_VEL
LIN {X 0,Y 277.284,Z 153.943,A -85,B 0,C 180,E1 -17514.341,E2 -17514.341} C_VEL
LIN {X 0,Y 277.244,Z 153.951,A -85,B 0,C 180,E1 -17517.836,E2 -17517.836} C_VEL
LIN {X 0,Y 277.29,Z 153.946,A -85,B 0,C 180,E1 -17521.212,E2 -17521.212} C_VEL
LIN {X 0,Y 277.315,Z 153.94,A -85,B 0,C 180,E1 -17524.479,E2 -17524.479} C_VEL
LIN {X 0,Y 277.281,Z 153.945,A -85,B 0,C 180,E1 -17527.654,E2 -17527.654} C_VEL
LIN {X 0,Y 277.32,Z 153.939,A -85,B 0,C 180,E1 -17530.764,E2 -17530.764} C_VEL
LIN {X 0,Y 277.408,Z 153.929,A -85,B 0,C 180,E1 -17535.324,E2 -17535.324} C_VEL
LIN {X 0,Y 277.505,Z 153.915,A -85,B 0,C 180,E1 -17539.788,E2 -17539.788} C_VEL
LIN {X 0,Y 277.648,Z 153.9,A -85,B 0,C 180,E1 -17542.728,E2 -17542.728} C_VEL
LIN {X 0,Y 277.82,Z 153.878,A -85,B 0,C 180,E1 -17548.55,E2 -17548.55} C_VEL
LIN {X 0,Y 277.82,Z 153.876,A -85,B 0,C 180,E1 -17551.449,E2 -17551.449} C_VEL
LIN {X 0,Y 277.647,Z 153.898,A -85,B 0,C 180,E1 -17557.27,E2 -17557.27} C_VEL
LIN {X 0,Y 277.505,Z 153.917,A -85,B 0,C 180,E1 -17560.211,E2 -17560.211} C_VEL
LIN {X 0,Y 277.432,Z 153.928,A -85,B 0,C 180,E1 -17564.674,E2 -17564.674} C_VEL
LIN {X 0,Y 277.342,Z 153.934,A -85,B 0,C 180,E1 -17569.233,E2 -17569.233} C_VEL
LIN {X 0,Y 277.289,Z 153.946,A -85,B 0,C 180,E1 -17574.158,E2 -17574.158} C_VEL
LIN {X 0,Y 277.332,Z 153.936,A -85,B 0,C 180,E1 -17577.509,E2 -17577.509} C_VEL
LIN {X 0,Y 277.269,Z 153.947,A -85,B 0,C 180,E1 -17580.481,E2 -17580.481} C_VEL
LIN {X 0,Y 277.252,Z 153.95,A -85,B 0,C 180,E1 -17583.894,E2 -17583.894} C_VEL
LIN {X 0,Y 277.286,Z 153.943,A -85,B 0,C 180,E1 -17587.466,E2 -17587.466} C_VEL
LIN {X 0,Y 277.261,Z 153.946,A -85,B 0,C 180,E1 -17591.226,E2 -17591.226} C_VEL
LIN {X 0,Y 277.247,Z 153.947,A -85,B 0,C 180,E1 -17595.216,E2 -17595.216} C_VEL
LIN {X 0,Y 277.284,Z 153.946,A -85,B 0,C 180,E1 -17599.496,E2 -17599.496} C_VEL
LIN {X 0,Y 277.284,Z 153.941,A -85,B 0,C 180,E1 -17602.534,E2 -17602.534} C_VEL
LIN {X 0,Y 277.251,Z 153.948,A -85,B 0,C 180,E1 -17606.106,E2 -17606.106} C_VEL
LIN {X 0,Y 277.258,Z 153.95,A -85,B 0,C 180,E1 -17609.539,E2 -17609.539} C_VEL
LIN {X 0,Y 277.358,Z 153.934,A -85,B 0,C 180,E1 -17612.865,E2 -17612.865} C_VEL
LIN {X 0,Y 277.326,Z 153.938,A -85,B 0,C 180,E1 -17616.08,E2 -17616.08} C_VEL
LIN {X 0,Y 277.343,Z 153.936,A -85,B 0,C 180,E1 -17620.767,E2 -17620.767} C_VEL
LIN {X 0,Y 277.432,Z 153.927,A -85,B 0,C 180,E1 -17625.326,E2 -17625.326} C_VEL
LIN {X 0,Y 277.442,Z 153.92,A -85,B 0,C 180,E1 -17628.969,E2 -17628.969} C_VEL
LIN {X 0,Y 276.821,Z 154.001,A -85,B 0,C 180,E1 -17630.182,E2 -17630.182} C_VEL
LIN {X 0,Y 273.999,Z 154.352,A -85,B 0,C 180,E1 -17632.158,E2 -17632.158} C_VEL
LIN {X 0,Y 271.569,Z 154.654,A -85,B 0,C 180,E1 -17633.765,E2 -17633.765} C_VEL
LIN {X 0,Y 270.513,Z 154.789,A -85,B 0,C 180,E1 -17635.01,E2 -17635.01} C_VEL
LIN {X 0,Y 270.421,Z 154.796,A -85,B 0,C 180,E1 -17635.432,E2 -17635.432} C_VEL
LIN {X 0,Y 270.786,Z 154.754,A -85,B 0,C 180,E1 -17638.513,E2 -17638.513} C_VEL
LIN {X 0,Y 270.786,Z 154.753,A -85,B 0,C 180,E1 -17641.488,E2 -17641.488} C_VEL
LIN {X 0,Y 270.61,Z 154.774,A -85,B 0,C 180,E1 -17647.462,E2 -17647.462} C_VEL
LIN {X 0,Y 270.44,Z 154.799,A -85,B 0,C 180,E1 -17650.482,E2 -17650.482} C_VEL
LIN {X 0,Y 270.402,Z 154.801,A -85,B 0,C 180,E1 -17655.065,E2 -17655.065} C_VEL
LIN {X 0,Y 270.3,Z 154.812,A -85,B 0,C 180,E1 -17659.756,E2 -17659.756} C_VEL
LIN {X 0,Y 270.237,Z 154.823,A -85,B 0,C 180,E1 -17664.59,E2 -17664.59} C_VEL
LIN {X 0,Y 270.271,Z 154.818,A -85,B 0,C 180,E1 -17667.909,E2 -17667.909} C_VEL
LIN {X 0,Y 270.184,Z 154.827,A -85,B 0,C 180,E1 -17671.349,E2 -17671.349} C_VEL
LIN {X 0,Y 270.216,Z 154.823,A -85,B 0,C 180,E1 -17674.904,E2 -17674.904} C_VEL
LIN {X 0,Y 270.222,Z 154.822,A -85,B 0,C 180,E1 -17678.718,E2 -17678.718} C_VEL
LIN {X 0,Y 270.192,Z 154.827,A -85,B 0,C 180,E1 -17682.555,E2 -17682.555} C_VEL
LIN {X 0,Y 270.165,Z 154.83,A -85,B 0,C 180,E1 -17686.752,E2 -17686.752} C_VEL
LIN {X 0,Y 270.175,Z 154.831,A -85,B 0,C 180,E1 -17689.435,E2 -17689.435} C_VEL
LIN {X 0,Y 270.228,Z 154.827,A -85,B 0,C 180,E1 -17693.731,E2 -17693.731} C_VEL
LIN {X 0,Y 270.308,Z 154.892,A -85,B 0,C 180,E1 -17695.973,E2 -17695.973} C_VEL
LIN {X 0,Y 273.404,Z 170.044,A -85,B 0,C 180,E1 -17700.765,E2 -17700.765} C_VEL
LIN {X 0,Y 274.428,Z 175.937,A -85,B 0,C 180,E1 -17702.551,E2 -17702.551} C_VEL
LIN {X 0,Y 273.905,Z 180.247,A -85,B 0,C 180,E1 -17703.775,E2 -17703.775} C_VEL
LIN {X 0,Y 278.961,Z 228.345,A -85,B 0,C 180,E1 -17705.79,E2 -17705.79} C_VEL
LIN {X 0,Y 276.856,Z 290.381,A -85,B 0,C 180,E1 -17707.864,E2 -17707.864} C_VEL
LIN {X 0,Y 275.933,Z 304.15,A -85,B 0,C 180,E1 -17708.621,E2 -17708.621} C_VEL
LIN {X 0,Y 274.808,Z 316.653,A -85,B 0,C 180,E1 -17709.608,E2 -17709.608} C_VEL
LIN {X 0,Y 273.569,Z 328.814,A -85,B 0,C 180,E1 -17710.881,E2 -17710.881} C_VEL
LIN {X 0,Y 272.307,Z 340.088,A -85,B 0,C 180,E1 -17712.386,E2 -17712.386} C_VEL
LIN {X 0,Y 270.977,Z 350.837,A -85,B 0,C 180,E1 -17714.198,E2 -17714.198} C_VEL
LIN {X 0,Y 270.107,Z 359.84,A -85,B 0,C 180,E1 -17716.074,E2 -17716.074} C_VEL
LIN {X 0,Y 269.341,Z 367.23,A -85,B 0,C 180,E1 -17717.952,E2 -17717.952} C_VEL
LIN {X 0,Y 268.791,Z 374.431,A -85,B 0,C 180,E1 -17720.215,E2 -17720.215} C_VEL
LIN {X 0,Y 268.514,Z 380.134,A -85,B 0,C 180,E1 -17722.481,E2 -17722.481} C_VEL
LIN {X 0,Y 268.509,Z 384.349,A -85,B 0,C 180,E1 -17724.627,E2 -17724.627} C_VEL
LIN {X 0,Y 268.427,Z 387.763,A -85,B 0,C 180,E1 -17726.999,E2 -17726.999} C_VEL
LIN {X 0,Y 268.48,Z 389.328,A -85,B 0,C 180,E1 -17728.501,E2 -17728.501} C_VEL
LIN {X 0,Y 268.621,Z 390.442,A -85,B 0,C 180,E1 -17730.001,E2 -17730.001} C_VEL
LIN {X 0,Y 268.312,Z 391.264,A -85,B 0,C 180,E1 -17733.003,E2 -17733.003} C_VEL
LIN {X 0,Y 268.194,Z 390.785,A -85,B 0,C 180,E1 -17735.255,E2 -17735.255} C_VEL
LIN {X 0,Y 268.34,Z 389.368,A -85,B 0,C 180,E1 -17737.525,E2 -17737.525} C_VEL
LIN {X 0,Y 268.642,Z 387.9,A -85,B 0,C 180,E1 -17739.031,E2 -17739.031} C_VEL
LIN {X 0,Y 269.29,Z 384.902,A -85,B 0,C 180,E1 -17741.288,E2 -17741.288} C_VEL
LIN {X 0,Y 270.337,Z 380.88,A -85,B 0,C 180,E1 -17743.532,E2 -17743.532} C_VEL
LIN {X 0,Y 271.962,Z 375.73,A -85,B 0,C 180,E1 -17745.745,E2 -17745.745} C_VEL
LIN {X 0,Y 273.702,Z 369.327,A -85,B 0,C 180,E1 -17747.947,E2 -17747.947} C_VEL
LIN {X 0,Y 276.131,Z 361.504,A -85,B 0,C 180,E1 -17750.097,E2 -17750.097} C_VEL
LIN {X 0,Y 279.022,Z 351.809,A -85,B 0,C 180,E1 -17752.199,E2 -17752.199} C_VEL
LIN {X 0,Y 281.762,Z 341.93,A -85,B 0,C 180,E1 -17753.912,E2 -17753.912} C_VEL
LIN {X 0,Y 284.516,Z 331.076,A -85,B 0,C 180,E1 -17755.417,E2 -17755.417} C_VEL
LIN {X 0,Y 287.159,Z 319.054,A -85,B 0,C 180,E1 -17756.726,E2 -17756.726} C_VEL
LIN {X 0,Y 289.632,Z 306.694,A -85,B 0,C 180,E1 -17757.749,E2 -17757.749} C_VEL
LIN {X 0,Y 291.563,Z 294.049,A -85,B 0,C 180,E1 -17758.527,E2 -17758.527} C_VEL
LIN {X 0,Y 293.005,Z 279.997,A -85,B 0,C 180,E1 -17759.134,E2 -17759.134} C_VEL
LIN {X 0,Y 296.319,Z 232.964,A -85,B 0,C 180,E1 -17760.717,E2 -17760.717} C_VEL
LIN {X 0,Y 295.031,Z 219.13,A -85,B 0,C 180,E1 -17761.633,E2 -17761.633} C_VEL
LIN {X 0,Y 293.308,Z 206.601,A -85,B 0,C 180,E1 -17762.621,E2 -17762.621} C_VEL
LIN {X 0,Y 292.439,Z 202.973,A -85,B 0,C 180,E1 -17762.992,E2 -17762.992} C_VEL
LIN {X 0,Y 287.892,Z 193.145,A -85,B 0,C 180,E1 -17764.555,E2 -17764.555} C_VEL
LIN {X 0,Y 284.85,Z 187.382,A -85,B 0,C 180,E1 -17765.638,E2 -17765.638} C_VEL
LIN {X 0,Y 282.434,Z 182.948,A -85,B 0,C 180,E1 -17766.556,E2 -17766.556} C_VEL
LIN {X 0,Y 279.346,Z 177.608,A -85,B 0,C 180,E1 -17767.79,E2 -17767.79} C_VEL
LIN {X 0,Y 276.114,Z 172.234,A -85,B 0,C 180,E1 -17769.194,E2 -17769.194} C_VEL
LIN {X 0,Y 274.042,Z 165.584,A -85,B 0,C 180,E1 -17773.038,E2 -17773.038} C_VEL
LIN {X 0,Y 272.488,Z 161.186,A -85,B 0,C 180,E1 -17776.235,E2 -17776.235} C_VEL
LIN {X 0,Y 271.093,Z 157.527,A -85,B 0,C 180,E1 -17779.599,E2 -17779.599} C_VEL
LIN {X 0,Y 270.225,Z 154.816,A -85,B 0,C 180,E1 -17782.793,E2 -17782.793} C_VEL
LIN {X 0,Y 270.206,Z 154.82,A -85,B 0,C 180,E1 -17786.892,E2 -17786.892} C_VEL
LIN {X 0,Y 270.223,Z 154.823,A -85,B 0,C 180,E1 -17790.385,E2 -17790.385} C_VEL
LIN {X 0,Y 270.265,Z 154.814,A -85,B 0,C 180,E1 -17793.763,E2 -17793.763} C_VEL
LIN {X 0,Y 270.236,Z 154.816,A -85,B 0,C 180,E1 -17797.038,E2 -17797.038} C_VEL
LIN {X 0,Y 270.296,Z 154.916,A -85,B 0,C 180,E1 -17799.398,E2 -17799.398} C_VEL
LIN {X 0,Y 271.576,Z 158.376,A -85,B 0,C 180,E1 -17803.461,E2 -17803.461} C_VEL
LIN {X 0,Y 271.92,Z 159.393,A -85,B 0,C 180,E1 -17804.314,E2 -17804.314} C_VEL
LIN {X 0,Y 275.585,Z 163.901,A -85,B 0,C 180,E1 -17806.062,E2 -17806.062} C_VEL
LIN {X 0,Y 280.587,Z 170.458,A -85,B 0,C 180,E1 -17808.159,E2 -17808.159} C_VEL
LIN {X 0,Y 286.313,Z 178.378,A -85,B 0,C 180,E1 -17810.255,E2 -17810.255} C_VEL
LIN {X 0,Y 292.872,Z 189.684,A -85,B 0,C 180,E1 -17812.458,E2 -17812.458} C_VEL
LIN {X 0,Y 297.059,Z 197.478,A -85,B 0,C 180,E1 -17813.737,E2 -17813.737} C_VEL
LIN {X 0,Y 298.318,Z 200.339,A -85,B 0,C 180,E1 -17814.135,E2 -17814.135} C_VEL
LIN {X 0,Y 293.527,Z 264.571,A -85,B 0,C 180,E1 -17816.353,E2 -17816.353} C_VEL
LIN {X 0,Y 292.178,Z 277.411,A -85,B 0,C 180,E1 -17817.07,E2 -17817.07} C_VEL
LIN {X 0,Y 290.611,Z 288.569,A -85,B 0,C 180,E1 -17817.921,E2 -17817.921} C_VEL
LIN {X 0,Y 288.473,Z 300.239,A -85,B 0,C 180,E1 -17819.069,E2 -17819.069} C_VEL
LIN {X 0,Y 285.945,Z 311.798,A -85,B 0,C 180,E1 -17820.528,E2 -17820.528} C_VEL
LIN {X 0,Y 283.32,Z 322.267,A -85,B 0,C 180,E1 -17822.191,E2 -17822.191} C_VEL
LIN {X 0,Y 280.837,Z 331.2,A -85,B 0,C 180,E1 -17823.976,E2 -17823.976} C_VEL
LIN {X 0,Y 278.081,Z 339.996,A -85,B 0,C 180,E1 -17826.166,E2 -17826.166} C_VEL
LIN {X 0,Y 275.67,Z 347.064,A -85,B 0,C 180,E1 -17828.439,E2 -17828.439} C_VEL
LIN {X 0,Y 273.351,Z 353.364,A -85,B 0,C 180,E1 -17831.066,E2 -17831.066} C_VEL
LIN {X 0,Y 271.722,Z 357.573,A -85,B 0,C 180,E1 -17833.46,E2 -17833.46} C_VEL
LIN {X 0,Y 270.395,Z 360.567,A -85,B 0,C 180,E1 -17835.909,E2 -17835.909} C_VEL
LIN {X 0,Y 269.446,Z 362.323,A -85,B 0,C 180,E1 -17838.239,E2 -17838.239} C_VEL
LIN {X 0,Y 268.968,Z 362.928,A -85,B 0,C 180,E1 -17839.857,E2 -17839.857} C_VEL
LIN {X 0,Y 268.606,Z 363.089,A -85,B 0,C 180,E1 -17841.487,E2 -17841.487} C_VEL
LIN {X 0,Y 268.314,Z 362.547,A -85,B 0,C 180,E1 -17843.542,E2 -17843.542} C_VEL
LIN {X 0,Y 268.194,Z 360.477,A -85,B 0,C 180,E1 -17846.454,E2 -17846.454} C_VEL
LIN {X 0,Y 268.391,Z 357.334,A -85,B 0,C 180,E1 -17848.975,E2 -17848.975} C_VEL
LIN {X 0,Y 268.802,Z 352.805,A -85,B 0,C 180,E1 -17851.527,E2 -17851.527} C_VEL
LIN {X 0,Y 269.356,Z 346.642,A -85,B 0,C 180,E1 -17854.122,E2 -17854.122} C_VEL
LIN {X 0,Y 270.025,Z 340.305,A -85,B 0,C 180,E1 -17856.211,E2 -17856.211} C_VEL
LIN {X 0,Y 271.013,Z 331.711,A -85,B 0,C 180,E1 -17858.489,E2 -17858.489} C_VEL
LIN {X 0,Y 272.047,Z 322.459,A -85,B 0,C 180,E1 -17860.471,E2 -17860.471} C_VEL
LIN {X 0,Y 273.152,Z 312.231,A -85,B 0,C 180,E1 -17862.234,E2 -17862.234} C_VEL
LIN {X 0,Y 274.27,Z 301.172,A -85,B 0,C 180,E1 -17863.777,E2 -17863.777} C_VEL
LIN {X 0,Y 275.374,Z 288.607,A -85,B 0,C 180,E1 -17865.15,E2 -17865.15} C_VEL
LIN {X 0,Y 276.419,Z 275.121,A -85,B 0,C 180,E1 -17866.257,E2 -17866.257} C_VEL
LIN {X 0,Y 277.037,Z 262.263,A -85,B 0,C 180,E1 -17867.008,E2 -17867.008} C_VEL
LIN {X 0,Y 277.786,Z 242.143,A -85,B 0,C 180,E1 -17867.733,E2 -17867.733} C_VEL
LIN {X 0,Y 279.873,Z 183.044,A -85,B 0,C 180,E1 -17869.653,E2 -17869.653} C_VEL
LIN {X 0,Y 274.87,Z 167.847,A -85,B 0,C 180,E1 -17870.504,E2 -17870.504} C_VEL
LIN {X 0,Y 270.246,Z 154.823,A -85,B 0,C 180,E1 -17871.276,E2 -17871.276} C_VEL
LIN {X 0,Y 270.201,Z 154.827,A -85,B 0,C 180,E1 -17875.094,E2 -17875.094} C_VEL
LIN {X 0,Y 270.2,Z 154.828,A -85,B 0,C 180,E1 -17879.13,E2 -17879.13} C_VEL
LIN {X 0,Y 270.265,Z 154.819,A -85,B 0,C 180,E1 -17882.145,E2 -17882.145} C_VEL
LIN {X 0,Y 270.277,Z 154.82,A -85,B 0,C 180,E1 -17885.518,E2 -17885.518} C_VEL
LIN {X 0,Y 270.27,Z 154.816,A -85,B 0,C 180,E1 -17890.242,E2 -17890.242} C_VEL
LIN {X 0,Y 270.367,Z 154.807,A -85,B 0,C 180,E1 -17894.933,E2 -17894.933} C_VEL
LIN {X 0,Y 270.44,Z 154.797,A -85,B 0,C 180,E1 -17899.518,E2 -17899.518} C_VEL
LIN {X 0,Y 270.606,Z 154.776,A -85,B 0,C 180,E1 -17902.538,E2 -17902.538} C_VEL
LIN {X 0,Y 270.786,Z 154.754,A -85,B 0,C 180,E1 -17908.512,E2 -17908.512} C_VEL
LIN {X 0,Y 270.786,Z 154.752,A -85,B 0,C 180,E1 -17911.487,E2 -17911.487} C_VEL
LIN {X 0,Y 270.606,Z 154.775,A -85,B 0,C 180,E1 -17917.461,E2 -17917.461} C_VEL
LIN {X 0,Y 270.44,Z 154.799,A -85,B 0,C 180,E1 -17920.481,E2 -17920.481} C_VEL
LIN {X 0,Y 270.401,Z 154.801,A -85,B 0,C 180,E1 -17925.064,E2 -17925.064} C_VEL
LIN {X 0,Y 270.299,Z 154.812,A -85,B 0,C 180,E1 -17929.755,E2 -17929.755} C_VEL
LIN {X 0,Y 270.235,Z 154.823,A -85,B 0,C 180,E1 -17934.589,E2 -17934.589} C_VEL
LIN {X 0,Y 270.272,Z 154.817,A -85,B 0,C 180,E1 -17937.908,E2 -17937.908} C_VEL
LIN {X 0,Y 270.182,Z 154.828,A -85,B 0,C 180,E1 -17941.348,E2 -17941.348} C_VEL
LIN {X 0,Y 270.213,Z 154.823,A -85,B 0,C 180,E1 -17944.903,E2 -17944.903} C_VEL
LIN {X 0,Y 270.219,Z 154.823,A -85,B 0,C 180,E1 -17948.717,E2 -17948.717} C_VEL
LIN {X 0,Y 270.219,Z 154.823,A -85,B 0,C 180,E1 -17952.548,E2 -17952.548} C_VEL
LIN {X 0,Y 270.2,Z 154.825,A -85,B 0,C 180,E1 -17956.742,E2 -17956.742} C_VEL
LIN {X 0,Y 270.234,Z 154.823,A -85,B 0,C 180,E1 -17959.446,E2 -17959.446} C_VEL
LIN {X 0,Y 270.253,Z 154.822,A -85,B 0,C 180,E1 -17963.722,E2 -17963.722} C_VEL
LIN {X 0,Y 270.201,Z 154.826,A -85,B 0,C 180,E1 -17966.893,E2 -17966.893} C_VEL
LIN {X 0,Y 270.226,Z 154.821,A -85,B 0,C 180,E1 -17970.387,E2 -17970.387} C_VEL
LIN {X 0,Y 270.262,Z 154.82,A -85,B 0,C 180,E1 -17973.764,E2 -17973.764} C_VEL
LIN {X 0,Y 270.23,Z 154.824,A -85,B 0,C 180,E1 -17977.039,E2 -17977.039} C_VEL
LIN {X 0,Y 270.299,Z 154.812,A -85,B 0,C 180,E1 -17980.245,E2 -17980.245} C_VEL
LIN {X 0,Y 270.4,Z 154.803,A -85,B 0,C 180,E1 -17984.936,E2 -17984.936} C_VEL
LIN {X 0,Y 270.439,Z 154.797,A -85,B 0,C 180,E1 -17989.519,E2 -17989.519} C_VEL
LIN {X 0,Y 270.605,Z 154.776,A -85,B 0,C 180,E1 -17992.539,E2 -17992.539} C_VEL
LIN {X 0,Y 270.421,Z 154.796,A -85,B 0,C 180,E1 -17995.432,E2 -17995.432} C_VEL
LIN {X 0,Y 269.794,Z 154.88,A -85,B 0,C 180,E1 -17996.678,E2 -17996.678} C_VEL
LIN {X 0,Y 267.149,Z 155.212,A -85,B 0,C 180,E1 -17998.716,E2 -17998.716} C_VEL
LIN {X 0,Y 264.046,Z 155.593,A -85,B 0,C 180,E1 -18001.218,E2 -18001.218} C_VEL
LIN {X 0,Y 263.661,Z 155.638,A -85,B 0,C 180,E1 -18002.08,E2 -18002.08} C_VEL
LIN {X 0,Y 263.571,Z 155.651,A -85,B 0,C 180,E1 -18007.662,E2 -18007.662} C_VEL
LIN {X 0,Y 263.373,Z 155.678,A -85,B 0,C 180,E1 -18010.766,E2 -18010.766} C_VEL
LIN {X 0,Y 263.35,Z 155.679,A -85,B 0,C 180,E1 -18015.479,E2 -18015.479} C_VEL
LIN {X 0,Y 263.262,Z 155.692,A -85,B 0,C 180,E1 -18020.307,E2 -18020.307} C_VEL
LIN {X 0,Y 263.192,Z 155.698,A -85,B 0,C 180,E1 -18025.294,E2 -18025.294} C_VEL
LIN {X 0,Y 263.179,Z 155.699,A -85,B 0,C 180,E1 -18028.73,E2 -18028.73} C_VEL
LIN {X 0,Y 263.133,Z 155.709,A -85,B 0,C 180,E1 -18032.289,E2 -18032.289} C_VEL
LIN {X 0,Y 263.19,Z 155.702,A -85,B 0,C 180,E1 -18035.978,E2 -18035.978} C_VEL
LIN {X 0,Y 263.14,Z 155.708,A -85,B 0,C 180,E1 -18039.867,E2 -18039.867} C_VEL
LIN {X 0,Y 263.128,Z 155.709,A -85,B 0,C 180,E1 -18043.984,E2 -18043.984} C_VEL
LIN {X 0,Y 263.125,Z 155.708,A -85,B 0,C 180,E1 -18048.407,E2 -18048.407} C_VEL
LIN {X 0,Y 263.185,Z 155.702,A -85,B 0,C 180,E1 -18053.237,E2 -18053.237} C_VEL
LIN {X 0,Y 263.267,Z 155.851,A -85,B 0,C 180,E1 -18055.696,E2 -18055.696} C_VEL
LIN {X 0,Y 266.33,Z 170.829,A -85,B 0,C 180,E1 -18060.554,E2 -18060.554} C_VEL
LIN {X 0,Y 267.346,Z 176.057,A -85,B 0,C 180,E1 -18062.186,E2 -18062.186} C_VEL
LIN {X 0,Y 267.043,Z 179.901,A -85,B 0,C 180,E1 -18063.319,E2 -18063.319} C_VEL
LIN {X 0,Y 272.091,Z 229.419,A -85,B 0,C 180,E1 -18065.439,E2 -18065.439} C_VEL
LIN {X 0,Y 269.967,Z 289.833,A -85,B 0,C 180,E1 -18067.521,E2 -18067.521} C_VEL
LIN {X 0,Y 269.084,Z 302.885,A -85,B 0,C 180,E1 -18068.251,E2 -18068.251} C_VEL
LIN {X 0,Y 267.923,Z 315.621,A -85,B 0,C 180,E1 -18069.261,E2 -18069.261} C_VEL
LIN {X 0,Y 266.649,Z 327.871,A -85,B 0,C 180,E1 -18070.565,E2 -18070.565} C_VEL
LIN {X 0,Y 265.371,Z 339.004,A -85,B 0,C 180,E1 -18072.07,E2 -18072.07} C_VEL
LIN {X 0,Y 264.064,Z 349.323,A -85,B 0,C 180,E1 -18073.824,E2 -18073.824} C_VEL
LIN {X 0,Y 263.169,Z 358.281,A -85,B 0,C 180,E1 -18075.699,E2 -18075.699} C_VEL
LIN {X 0,Y 262.382,Z 365.858,A -85,B 0,C 180,E1 -18077.627,E2 -18077.627} C_VEL
LIN {X 0,Y 261.757,Z 373.282,A -85,B 0,C 180,E1 -18079.95,E2 -18079.95} C_VEL
LIN {X 0,Y 261.474,Z 379.143,A -85,B 0,C 180,E1 -18082.277,E2 -18082.277} C_VEL
LIN {X 0,Y 261.445,Z 383.752,A -85,B 0,C 180,E1 -18084.638,E2 -18084.638} C_VEL
LIN {X 0,Y 261.361,Z 387.039,A -85,B 0,C 180,E1 -18086.918,E2 -18086.918} C_VEL
LIN {X 0,Y 261.399,Z 388.663,A -85,B 0,C 180,E1 -18088.46,E2 -18088.46} C_VEL
LIN {X 0,Y 261.554,Z 389.857,A -85,B 0,C 180,E1 -18090.001,E2 -18090.001} C_VEL
LIN {X 0,Y 261.269,Z 390.559,A -85,B 0,C 180,E1 -18091.542,E2 -18091.542} C_VEL
LIN {X 0,Y 261.236,Z 390.826,A -85,B 0,C 180,E1 -18093.085,E2 -18093.085} C_VEL
LIN {X 0,Y 261.144,Z 390.13,A -85,B 0,C 180,E1 -18096.18,E2 -18096.18} C_VEL
LIN {X 0,Y 261.288,Z 389.165,A -85,B 0,C 180,E1 -18097.73,E2 -18097.73} C_VEL
LIN {X 0,Y 261.588,Z 387.763,A -85,B 0,C 180,E1 -18099.277,E2 -18099.277} C_VEL
LIN {X 0,Y 262.303,Z 384.888,A -85,B 0,C 180,E1 -18101.593,E2 -18101.593} C_VEL
LIN {X 0,Y 263.437,Z 380.993,A -85,B 0,C 180,E1 -18103.893,E2 -18103.893} C_VEL
LIN {X 0,Y 265.137,Z 376.001,A -85,B 0,C 180,E1 -18106.161,E2 -18106.161} C_VEL
LIN {X 0,Y 266.975,Z 369.816,A -85,B 0,C 180,E1 -18108.415,E2 -18108.415} C_VEL
LIN {X 0,Y 269.503,Z 362.182,A -85,B 0,C 180,E1 -18110.613,E2 -18110.613} C_VEL
LIN {X 0,Y 272.539,Z 352.794,A -85,B 0,C 180,E1 -18112.756,E2 -18112.756} C_VEL
LIN {X 0,Y 275.689,Z 342.153,A -85,B 0,C 180,E1 -18114.674,E2 -18114.674} C_VEL
LIN {X 0,Y 278.584,Z 331.562,A -85,B 0,C 180,E1 -18116.199,E2 -18116.199} C_VEL
LIN {X 0,Y 281.333,Z 319.905,A -85,B 0,C 180,E1 -18117.526,E2 -18117.526} C_VEL
LIN {X 0,Y 284.103,Z 306.809,A -85,B 0,C 180,E1 -18118.639,E2 -18118.639} C_VEL
LIN {X 0,Y 286.111,Z 294.459,A -85,B 0,C 180,E1 -18119.425,E2 -18119.425} C_VEL
LIN {X 0,Y 287.675,Z 280.28,A -85,B 0,C 180,E1 -18120.055,E2 -18120.055} C_VEL
LIN {X 0,Y 291.208,Z 234.024,A -85,B 0,C 180,E1 -18121.655,E2 -18121.655} C_VEL
LIN {X 0,Y 289.888,Z 219.289,A -85,B 0,C 180,E1 -18122.681,E2 -18122.681} C_VEL
LIN {X 0,Y 288.24,Z 207.721,A -85,B 0,C 180,E1 -18123.655,E2 -18123.655} C_VEL
LIN {X 0,Y 284.359,Z 198.732,A -85,B 0,C 180,E1 -18125.103,E2 -18125.103} C_VEL
LIN {X 0,Y 280.254,Z 190.577,A -85,B 0,C 180,E1 -18126.687,E2 -18126.687} C_VEL
LIN {X 0,Y 275.996,Z 183.023,A -85,B 0,C 180,E1 -18128.461,E2 -18128.461} C_VEL
LIN {X 0,Y 272.504,Z 177.159,A -85,B 0,C 180,E1 -18130.084,E2 -18130.084} C_VEL
LIN {X 0,Y 268.956,Z 171.76,A -85,B 0,C 180,E1 -18131.905,E2 -18131.905} C_VEL
LIN {X 0,Y 268.474,Z 170.734,A -85,B 0,C 180,E1 -18132.253,E2 -18132.253} C_VEL
LIN {X 0,Y 267.005,Z 166.44,A -85,B 0,C 180,E1 -18135.291,E2 -18135.291} C_VEL
LIN {X 0,Y 265.704,Z 162.626,A -85,B 0,C 180,E1 -18138.603,E2 -18138.603} C_VEL
LIN {X 0,Y 264.496,Z 158.986,A -85,B 0,C 180,E1 -18142.859,E2 -18142.859} C_VEL
LIN {X 0,Y 263.395,Z 156.91,A -85,B 0,C 180,E1 -18147.747,E2 -18147.747} C_VEL
LIN {X 0,Y 263.32,Z 156.446,A -85,B 0,C 180,E1 -18151.287,E2 -18151.287} C_VEL
LIN {X 0,Y 263.545,Z 157.092,A -85,B 0,C 180,E1 -18155.052,E2 -18155.052} C_VEL
LIN {X 0,Y 264.595,Z 159.403,A -85,B 0,C 180,E1 -18159.799,E2 -18159.799} C_VEL
LIN {X 0,Y 265.055,Z 160.739,A -85,B 0,C 180,E1 -18161.296,E2 -18161.296} C_VEL
LIN {X 0,Y 269.201,Z 165.448,A -85,B 0,C 180,E1 -18163.708,E2 -18163.708} C_VEL
LIN {X 0,Y 274.012,Z 171.579,A -85,B 0,C 180,E1 -18166.088,E2 -18166.088} C_VEL
LIN {X 0,Y 277.875,Z 176.873,A -85,B 0,C 180,E1 -18167.769,E2 -18167.769} C_VEL
LIN {X 0,Y 282.881,Z 183.945,A -85,B 0,C 180,E1 -18169.686,E2 -18169.686} C_VEL
LIN {X 0,Y 289.309,Z 195.351,A -85,B 0,C 180,E1 -18171.962,E2 -18171.962} C_VEL
LIN {X 0,Y 293.208,Z 202.946,A -85,B 0,C 180,E1 -18173.22,E2 -18173.22} C_VEL
LIN {X 0,Y 288.31,Z 264.527,A -85,B 0,C 180,E1 -18175.399,E2 -18175.399} C_VEL
LIN {X 0,Y 286.838,Z 277.629,A -85,B 0,C 180,E1 -18176.136,E2 -18176.136} C_VEL
LIN {X 0,Y 285.19,Z 288.857,A -85,B 0,C 180,E1 -18176.998,E2 -18176.998} C_VEL
LIN {X 0,Y 282.847,Z 301.088,A -85,B 0,C 180,E1 -18178.22,E2 -18178.22} C_VEL
LIN {X 0,Y 280.199,Z 312.551,A -85,B 0,C 180,E1 -18179.694,E2 -18179.694} C_VEL
LIN {X 0,Y 277.568,Z 322.3,A -85,B 0,C 180,E1 -18181.269,E2 -18181.269} C_VEL
LIN {X 0,Y 274.559,Z 332.353,A -85,B 0,C 180,E1 -18183.333,E2 -18183.333} C_VEL
LIN {X 0,Y 272.1,Z 339.683,A -85,B 0,C 180,E1 -18185.186,E2 -18185.186} C_VEL
LIN {X 0,Y 269.524,Z 346.923,A -85,B 0,C 180,E1 -18187.491,E2 -18187.491} C_VEL
LIN {X 0,Y 267.276,Z 352.625,A -85,B 0,C 180,E1 -18189.841,E2 -18189.841} C_VEL
LIN {X 0,Y 265.421,Z 357.021,A -85,B 0,C 180,E1 -18192.229,E2 -18192.229} C_VEL
LIN {X 0,Y 264.407,Z 359.315,A -85,B 0,C 180,E1 -18193.84,E2 -18193.84} C_VEL
LIN {X 0,Y 263.242,Z 361.582,A -85,B 0,C 180,E1 -18196.027,E2 -18196.027} C_VEL
LIN {X 0,Y 262.187,Z 363.204,A -85,B 0,C 180,E1 -18198.763,E2 -18198.763} C_VEL
LIN {X 0,Y 261.733,Z 363.511,A -85,B 0,C 180,E1 -18200.43,E2 -18200.43} C_VEL
LIN {X 0,Y 261.395,Z 363.357,A -85,B 0,C 180,E1 -18202.111,E2 -18202.111} C_VEL
LIN {X 0,Y 261.206,Z 362.702,A -85,B 0,C 180,E1 -18203.821,E2 -18203.821} C_VEL
LIN {X 0,Y 261.087,Z 361.526,A -85,B 0,C 180,E1 -18205.511,E2 -18205.511} C_VEL
LIN {X 0,Y 261.207,Z 358.758,A -85,B 0,C 180,E1 -18208.09,E2 -18208.09} C_VEL
LIN {X 0,Y 261.592,Z 354.631,A -85,B 0,C 180,E1 -18210.714,E2 -18210.714} C_VEL
LIN {X 0,Y 262.031,Z 349.485,A -85,B 0,C 180,E1 -18213.131,E2 -18213.131} C_VEL
LIN {X 0,Y 262.7,Z 342.782,A -85,B 0,C 180,E1 -18215.582,E2 -18215.582} C_VEL
LIN {X 0,Y 263.55,Z 335.089,A -85,B 0,C 180,E1 -18217.83,E2 -18217.83} C_VEL
LIN {X 0,Y 264.676,Z 325.425,A -85,B 0,C 180,E1 -18220.084,E2 -18220.084} C_VEL
LIN {X 0,Y 265.858,Z 314.661,A -85,B 0,C 180,E1 -18222.094,E2 -18222.094} C_VEL
LIN {X 0,Y 267.054,Z 303.9,A -85,B 0,C 180,E1 -18223.694,E2 -18223.694} C_VEL
LIN {X 0,Y 268.171,Z 291.408,A -85,B 0,C 180,E1 -18225.172,E2 -18225.172} C_VEL
LIN {X 0,Y 269.203,Z 279.021,A -85,B 0,C 180,E1 -18226.288,E2 -18226.288} C_VEL
LIN {X 0,Y 269.982,Z 264.911,A -85,B 0,C 180,E1 -18227.212,E2 -18227.212} C_VEL
LIN {X 0,Y 270.615,Z 250.647,A -85,B 0,C 180,E1 -18227.804,E2 -18227.804} C_VEL
LIN {X 0,Y 273.071,Z 184.398,A -85,B 0,C 180,E1 -18230.027,E2 -18230.027} C_VEL
LIN {X 0,Y 268.029,Z 169.322,A -85,B 0,C 180,E1 -18230.895,E2 -18230.895} C_VEL
LIN {X 0,Y 263.189,Z 155.703,A -85,B 0,C 180,E1 -18231.743,E2 -18231.743} C_VEL
LIN {X 0,Y 263.167,Z 155.704,A -85,B 0,C 180,E1 -18235.887,E2 -18235.887} C_VEL
LIN {X 0,Y 263.151,Z 155.709,A -85,B 0,C 180,E1 -18239.506,E2 -18239.506} C_VEL
LIN {X 0,Y 263.194,Z 155.702,A -85,B 0,C 180,E1 -18243.002,E2 -18243.002} C_VEL
LIN {X 0,Y 263.182,Z 155.7,A -85,B 0,C 180,E1 -18246.386,E2 -18246.386} C_VEL
LIN {X 0,Y 263.25,Z 155.692,A -85,B 0,C 180,E1 -18249.692,E2 -18249.692} C_VEL
LIN {X 0,Y 263.309,Z 155.684,A -85,B 0,C 180,E1 -18254.519,E2 -18254.519} C_VEL
LIN {X 0,Y 263.373,Z 155.679,A -85,B 0,C 180,E1 -18259.234,E2 -18259.234} C_VEL
LIN {X 0,Y 263.568,Z 155.652,A -85,B 0,C 180,E1 -18262.338,E2 -18262.338} C_VEL
LIN {X 0,Y 263.75,Z 155.63,A -85,B 0,C 180,E1 -18268.473,E2 -18268.473} C_VEL
LIN {X 0,Y 263.75,Z 155.628,A -85,B 0,C 180,E1 -18271.526,E2 -18271.526} C_VEL
LIN {X 0,Y 263.568,Z 155.651,A -85,B 0,C 180,E1 -18277.661,E2 -18277.661} C_VEL
LIN {X 0,Y 263.372,Z 155.677,A -85,B 0,C 180,E1 -18280.765,E2 -18280.765} C_VEL
LIN {X 0,Y 263.349,Z 155.679,A -85,B 0,C 180,E1 -18285.478,E2 -18285.478} C_VEL
LIN {X 0,Y 263.26,Z 155.692,A -85,B 0,C 180,E1 -18290.306,E2 -18290.306} C_VEL
LIN {X 0,Y 263.191,Z 155.698,A -85,B 0,C 180,E1 -18295.292,E2 -18295.292} C_VEL
LIN {X 0,Y 263.181,Z 155.7,A -85,B 0,C 180,E1 -18298.729,E2 -18298.729} C_VEL
LIN {X 0,Y 263.131,Z 155.709,A -85,B 0,C 180,E1 -18302.288,E2 -18302.288} C_VEL
LIN {X 0,Y 263.187,Z 155.701,A -85,B 0,C 180,E1 -18305.977,E2 -18305.977} C_VEL
LIN {X 0,Y 263.157,Z 155.706,A -85,B 0,C 180,E1 -18309.862,E2 -18309.862} C_VEL
LIN {X 0,Y 263.142,Z 155.706,A -85,B 0,C 180,E1 -18313.979,E2 -18313.979} C_VEL
LIN {X 0,Y 263.147,Z 155.705,A -85,B 0,C 180,E1 -18318.4,E2 -18318.4} C_VEL
LIN {X 0,Y 263.185,Z 155.699,A -85,B 0,C 180,E1 -18322.108,E2 -18322.108} C_VEL
LIN {X 0,Y 263.18,Z 155.702,A -85,B 0,C 180,E1 -18325.891,E2 -18325.891} C_VEL
LIN {X 0,Y 263.148,Z 155.707,A -85,B 0,C 180,E1 -18329.507,E2 -18329.507} C_VEL
LIN {X 0,Y 263.191,Z 155.699,A -85,B 0,C 180,E1 -18333.003,E2 -18333.003} C_VEL
LIN {X 0,Y 263.181,Z 155.699,A -85,B 0,C 180,E1 -18336.387,E2 -18336.387} C_VEL
LIN {X 0,Y 263.261,Z 155.69,A -85,B 0,C 180,E1 -18339.694,E2 -18339.694} C_VEL
LIN {X 0,Y 263.348,Z 155.679,A -85,B 0,C 180,E1 -18344.522,E2 -18344.522} C_VEL
LIN {X 0,Y 263.372,Z 155.679,A -85,B 0,C 180,E1 -18349.235,E2 -18349.235} C_VEL
LIN {X 0,Y 263.567,Z 155.652,A -85,B 0,C 180,E1 -18352.339,E2 -18352.339} C_VEL
LIN {X 0,Y 263.75,Z 155.63,A -85,B 0,C 180,E1 -18358.474,E2 -18358.474} C_VEL
LIN {X 0,Y 263.75,Z 155.629,A -85,B 0,C 180,E1 -18361.527,E2 -18361.527} C_VEL
LIN {X 0,Y 263.661,Z 155.638,A -85,B 0,C 180,E1 -18362.08,E2 -18362.08} C_VEL
LIN {X 0,Y 262.874,Z 155.738,A -85,B 0,C 180,E1 -18363.354,E2 -18363.354} C_VEL
LIN {X 0,Y 259.977,Z 156.098,A -85,B 0,C 180,E1 -18365.43,E2 -18365.43} C_VEL
LIN {X 0,Y 257.589,Z 156.398,A -85,B 0,C 180,E1 -18367.119,E2 -18367.119} C_VEL
LIN {X 0,Y 256.572,Z 156.525,A -85,B 0,C 180,E1 -18368.428,E2 -18368.428} C_VEL
LIN {X 0,Y 256.488,Z 156.531,A -85,B 0,C 180,E1 -18368.872,E2 -18368.872} C_VEL
LIN {X 0,Y 256.294,Z 156.56,A -85,B 0,C 180,E1 -18372.673,E2 -18372.673} C_VEL
LIN {X 0,Y 256.282,Z 156.562,A -85,B 0,C 180,E1 -18376.303,E2 -18376.303} C_VEL
LIN {X 0,Y 256.152,Z 156.574,A -85,B 0,C 180,E1 -18381.118,E2 -18381.118} C_VEL
LIN {X 0,Y 256.17,Z 156.573,A -85,B 0,C 180,E1 -18385.131,E2 -18385.131} C_VEL
LIN {X 0,Y 256.113,Z 156.579,A -85,B 0,C 180,E1 -18389.6,E2 -18389.6} C_VEL
LIN {X 0,Y 256.085,Z 156.584,A -85,B 0,C 180,E1 -18393.291,E2 -18393.291} C_VEL
LIN {X 0,Y 256.141,Z 156.575,A -85,B 0,C 180,E1 -18397.279,E2 -18397.279} C_VEL
LIN {X 0,Y 256.085,Z 156.584,A -85,B 0,C 180,E1 -18401.198,E2 -18401.198} C_VEL
LIN {X 0,Y 256.059,Z 156.587,A -85,B 0,C 180,E1 -18405.531,E2 -18405.531} C_VEL
LIN {X 0,Y 256.055,Z 156.588,A -85,B 0,C 180,E1 -18408.797,E2 -18408.797} C_VEL
LIN {X 0,Y 256.133,Z 156.58,A -85,B 0,C 180,E1 -18412.869,E2 -18412.869} C_VEL
LIN {X 0,Y 256.224,Z 156.712,A -85,B 0,C 180,E1 -18415.375,E2 -18415.375} C_VEL
LIN {X 0,Y 259.159,Z 171.19,A -85,B 0,C 180,E1 -18420.204,E2 -18420.204} C_VEL
LIN {X 0,Y 260.348,Z 177.565,A -85,B 0,C 180,E1 -18422.248,E2 -18422.248} C_VEL
LIN {X 0,Y 260.194,Z 179.524,A -85,B 0,C 180,E1 -18422.841,E2 -18422.841} C_VEL
LIN {X 0,Y 264.988,Z 227.231,A -85,B 0,C 180,E1 -18424.961,E2 -18424.961} C_VEL
LIN {X 0,Y 265.188,Z 230.182,A -85,B 0,C 180,E1 -18425.081,E2 -18425.081} C_VEL
LIN {X 0,Y 263.029,Z 289.62,A -85,B 0,C 180,E1 -18427.206,E2 -18427.206} C_VEL
LIN {X 0,Y 262.145,Z 302.612,A -85,B 0,C 180,E1 -18427.956,E2 -18427.956} C_VEL
LIN {X 0,Y 261.042,Z 314.301,A -85,B 0,C 180,E1 -18428.895,E2 -18428.895} C_VEL
LIN {X 0,Y 259.735,Z 326.749,A -85,B 0,C 180,E1 -18430.232,E2 -18430.232} C_VEL
LIN {X 0,Y 258.434,Z 338.01,A -85,B 0,C 180,E1 -18431.776,E2 -18431.776} C_VEL
LIN {X 0,Y 257.134,Z 348.015,A -85,B 0,C 180,E1 -18433.486,E2 -18433.486} C_VEL
LIN {X 0,Y 256.06,Z 358.343,A -85,B 0,C 180,E1 -18435.699,E2 -18435.699} C_VEL
LIN {X 0,Y 255.273,Z 365.849,A -85,B 0,C 180,E1 -18437.681,E2 -18437.681} C_VEL
LIN {X 0,Y 254.672,Z 373.19,A -85,B 0,C 180,E1 -18440.069,E2 -18440.069} C_VEL
LIN {X 0,Y 254.409,Z 378.123,A -85,B 0,C 180,E1 -18442.061,E2 -18442.061} C_VEL
LIN {X 0,Y 254.379,Z 382.112,A -85,B 0,C 180,E1 -18444.053,E2 -18444.053} C_VEL
LIN {X 0,Y 254.347,Z 385.258,A -85,B 0,C 180,E1 -18446.04,E2 -18446.04} C_VEL
LIN {X 0,Y 254.318,Z 387.998,A -85,B 0,C 180,E1 -18448.417,E2 -18448.417} C_VEL
LIN {X 0,Y 254.487,Z 389.25,A -85,B 0,C 180,E1 -18450.001,E2 -18450.001} C_VEL
LIN {X 0,Y 254.191,Z 390.031,A -85,B 0,C 180,E1 -18451.585,E2 -18451.585} C_VEL
LIN {X 0,Y 254.16,Z 390.386,A -85,B 0,C 180,E1 -18453.171,E2 -18453.171} C_VEL
LIN {X 0,Y 254.055,Z 389.81,A -85,B 0,C 180,E1 -18456.354,E2 -18456.354} C_VEL
LIN {X 0,Y 254.231,Z 388.929,A -85,B 0,C 180,E1 -18457.945,E2 -18457.945} C_VEL
LIN {X 0,Y 254.552,Z 387.626,A -85,B 0,C 180,E1 -18459.536,E2 -18459.536} C_VEL
LIN {X 0,Y 255.622,Z 383.722,A -85,B 0,C 180,E1 -18462.707,E2 -18462.707} C_VEL
LIN {X 0,Y 257.12,Z 379.637,A -85,B 0,C 180,E1 -18465.051,E2 -18465.051} C_VEL
LIN {X 0,Y 259.334,Z 373.473,A -85,B 0,C 180,E1 -18467.751,E2 -18467.751} C_VEL
LIN {X 0,Y 261.538,Z 366.781,A -85,B 0,C 180,E1 -18470.036,E2 -18470.036} C_VEL
LIN {X 0,Y 264.479,Z 358.561,A -85,B 0,C 180,E1 -18472.252,E2 -18472.252} C_VEL
LIN {X 0,Y 267.784,Z 348.532,A -85,B 0,C 180,E1 -18474.417,E2 -18474.417} C_VEL
LIN {X 0,Y 271.035,Z 338.146,A -85,B 0,C 180,E1 -18476.156,E2 -18476.156} C_VEL
LIN {X 0,Y 274.119,Z 326.715,A -85,B 0,C 180,E1 -18477.691,E2 -18477.691} C_VEL
LIN {X 0,Y 276.776,Z 315.704,A -85,B 0,C 180,E1 -18478.846,E2 -18478.846} C_VEL
LIN {X 0,Y 279.449,Z 302.671,A -85,B 0,C 180,E1 -18479.886,E2 -18479.886} C_VEL
LIN {X 0,Y 281.631,Z 289.146,A -85,B 0,C 180,E1 -18480.665,E2 -18480.665} C_VEL
LIN {X 0,Y 283.314,Z 271.61,A -85,B 0,C 180,E1 -18481.343,E2 -18481.343} C_VEL
LIN {X 0,Y 286.192,Z 234.894,A -85,B 0,C 180,E1 -18482.648,E2 -18482.648} C_VEL
LIN {X 0,Y 284.991,Z 220.878,A -85,B 0,C 180,E1 -18483.678,E2 -18483.678} C_VEL
LIN {X 0,Y 283.778,Z 211.326,A -85,B 0,C 180,E1 -18484.513,E2 -18484.513} C_VEL
LIN {X 0,Y 279.743,Z 202.004,A -85,B 0,C 180,E1 -18486.106,E2 -18486.106} C_VEL
LIN {X 0,Y 275.96,Z 194.319,A -85,B 0,C 180,E1 -18487.698,E2 -18487.698} C_VEL
LIN {X 0,Y 272.936,Z 188.792,A -85,B 0,C 180,E1 -18489.057,E2 -18489.057} C_VEL
LIN {X 0,Y 269.542,Z 182.97,A -85,B 0,C 180,E1 -18490.715,E2 -18490.715} C_VEL
LIN {X 0,Y 265.405,Z 176.365,A -85,B 0,C 180,E1 -18493.025,E2 -18493.025} C_VEL
LIN {X 0,Y 260.738,Z 169.217,A -85,B 0,C 180,E1 -18496.328,E2 -18496.328} C_VEL
LIN {X 0,Y 259.581,Z 165.946,A -85,B 0,C 180,E1 -18499.474,E2 -18499.474} C_VEL
LIN {X 0,Y 258.635,Z 162.978,A -85,B 0,C 180,E1 -18503.286,E2 -18503.286} C_VEL
LIN {X 0,Y 257.727,Z 161.199,A -85,B 0,C 180,E1 -18507.71,E2 -18507.71} C_VEL
LIN {X 0,Y 257.639,Z 160.72,A -85,B 0,C 180,E1 -18510.8,E2 -18510.8} C_VEL
LIN {X 0,Y 257.766,Z 161.122,A -85,B 0,C 180,E1 -18514.135,E2 -18514.135} C_VEL
LIN {X 0,Y 258.231,Z 162.281,A -85,B 0,C 180,E1 -18517.106,E2 -18517.106} C_VEL
LIN {X 0,Y 263.119,Z 167.541,A -85,B 0,C 180,E1 -18521.001,E2 -18521.001} C_VEL
LIN {X 0,Y 267.533,Z 172.776,A -85,B 0,C 180,E1 -18523.65,E2 -18523.65} C_VEL
LIN {X 0,Y 271.249,Z 177.638,A -85,B 0,C 180,E1 -18525.563,E2 -18525.563} C_VEL
LIN {X 0,Y 274.881,Z 182.733,A -85,B 0,C 180,E1 -18527.217,E2 -18527.217} C_VEL
LIN {X 0,Y 279.039,Z 188.742,A -85,B 0,C 180,E1 -18528.902,E2 -18528.902} C_VEL
LIN {X 0,Y 283.185,Z 196.214,A -85,B 0,C 180,E1 -18530.514,E2 -18530.514} C_VEL
LIN {X 0,Y 287.78,Z 204.983,A -85,B 0,C 180,E1 -18532.143,E2 -18532.143} C_VEL
LIN {X 0,Y 288.232,Z 206.331,A -85,B 0,C 180,E1 -18532.325,E2 -18532.325} C_VEL
LIN {X 0,Y 283.214,Z 265.168,A -85,B 0,C 180,E1 -18534.42,E2 -18534.42} C_VEL
LIN {X 0,Y 281.742,Z 277.493,A -85,B 0,C 180,E1 -18535.115,E2 -18535.115} C_VEL
LIN {X 0,Y 279.89,Z 289.358,A -85,B 0,C 180,E1 -18536.04,E2 -18536.04} C_VEL
LIN {X 0,Y 277.411,Z 301.491,A -85,B 0,C 180,E1 -18537.277,E2 -18537.277} C_VEL
LIN {X 0,Y 274.437,Z 313.575,A -85,B 0,C 180,E1 -18538.859,E2 -18538.859} C_VEL
LIN {X 0,Y 271.854,Z 322.718,A -85,B 0,C 180,E1 -18540.37,E2 -18540.37} C_VEL
LIN {X 0,Y 268.947,Z 331.855,A -85,B 0,C 180,E1 -18542.246,E2 -18542.246} C_VEL
LIN {X 0,Y 265.761,Z 340.783,A -85,B 0,C 180,E1 -18544.55,E2 -18544.55} C_VEL
LIN {X 0,Y 263.103,Z 347.642,A -85,B 0,C 180,E1 -18546.831,E2 -18546.831} C_VEL
LIN {X 0,Y 260.625,Z 353.464,A -85,B 0,C 180,E1 -18549.311,E2 -18549.311} C_VEL
LIN {X 0,Y 258.558,Z 357.979,A -85,B 0,C 180,E1 -18551.89,E2 -18551.89} C_VEL
LIN {X 0,Y 257.108,Z 360.894,A -85,B 0,C 180,E1 -18554.241,E2 -18554.241} C_VEL
LIN {X 0,Y 256.103,Z 362.539,A -85,B 0,C 180,E1 -18556.161,E2 -18556.161} C_VEL
LIN {X 0,Y 254.935,Z 363.884,A -85,B 0,C 180,E1 -18559.318,E2 -18559.318} C_VEL
LIN {X 0,Y 254.507,Z 363.922,A -85,B 0,C 180,E1 -18561.037,E2 -18561.037} C_VEL
LIN {X 0,Y 254.075,Z 362.762,A -85,B 0,C 180,E1 -18564.101,E2 -18564.101} C_VEL
LIN {X 0,Y 253.991,Z 360.997,A -85,B 0,C 180,E1 -18566.277,E2 -18566.277} C_VEL
LIN {X 0,Y 254.192,Z 357.717,A -85,B 0,C 180,E1 -18568.936,E2 -18568.936} C_VEL
LIN {X 0,Y 254.65,Z 353.053,A -85,B 0,C 180,E1 -18571.625,E2 -18571.625} C_VEL
LIN {X 0,Y 255.223,Z 346.84,A -85,B 0,C 180,E1 -18574.299,E2 -18574.299} C_VEL
LIN {X 0,Y 255.966,Z 339.811,A -85,B 0,C 180,E1 -18576.668,E2 -18576.668} C_VEL
LIN {X 0,Y 256.962,Z 331.285,A -85,B 0,C 180,E1 -18578.98,E2 -18578.98} C_VEL
LIN {X 0,Y 258.127,Z 321.698,A -85,B 0,C 180,E1 -18581.059,E2 -18581.059} C_VEL
LIN {X 0,Y 259.344,Z 310.795,A -85,B 0,C 180,E1 -18582.972,E2 -18582.972} C_VEL
LIN {X 0,Y 260.482,Z 299.525,A -85,B 0,C 180,E1 -18584.547,E2 -18584.547} C_VEL
LIN {X 0,Y 261.663,Z 286.518,A -85,B 0,C 180,E1 -18585.966,E2 -18585.966} C_VEL
LIN {X 0,Y 262.607,Z 274.339,A -85,B 0,C 180,E1 -18586.965,E2 -18586.965} C_VEL
LIN {X 0,Y 263.292,Z 260.792,A -85,B 0,C 180,E1 -18587.757,E2 -18587.757} C_VEL
LIN {X 0,Y 266.15,Z 185.461,A -85,B 0,C 180,E1 -18590.416,E2 -18590.416} C_VEL
LIN {X 0,Y 261.18,Z 170.829,A -85,B 0,C 180,E1 -18591.292,E2 -18591.292} C_VEL
LIN {X 0,Y 256.151,Z 156.577,A -85,B 0,C 180,E1 -18592.214,E2 -18592.214} C_VEL
LIN {X 0,Y 256.076,Z 156.585,A -85,B 0,C 180,E1 -18596.708,E2 -18596.708} C_VEL
LIN {X 0,Y 256.139,Z 156.583,A -85,B 0,C 180,E1 -18601.404,E2 -18601.404} C_VEL
LIN {X 0,Y 256.166,Z 156.576,A -85,B 0,C 180,E1 -18605.698,E2 -18605.698} C_VEL
LIN {X 0,Y 256.161,Z 156.578,A -85,B 0,C 180,E1 -18609.104,E2 -18609.104} C_VEL
LIN {X 0,Y 256.243,Z 156.564,A -85,B 0,C 180,E1 -18614.081,E2 -18614.081} C_VEL
LIN {X 0,Y 256.288,Z 156.56,A -85,B 0,C 180,E1 -18617.327,E2 -18617.327} C_VEL
LIN {X 0,Y 256.479,Z 156.536,A -85,B 0,C 180,E1 -18620.56,E2 -18620.56} C_VEL
LIN {X 0,Y 256.484,Z 156.533,A -85,B 0,C 180,E1 -18623.707,E2 -18623.707} C_VEL
LIN {X 0,Y 256.713,Z 156.507,A -85,B 0,C 180,E1 -18628.431,E2 -18628.431} C_VEL
LIN {X 0,Y 256.713,Z 156.504,A -85,B 0,C 180,E1 -18631.568,E2 -18631.568} C_VEL
LIN {X 0,Y 256.536,Z 156.528,A -85,B 0,C 180,E1 -18637.872,E2 -18637.872} C_VEL
LIN {X 0,Y 256.308,Z 156.555,A -85,B 0,C 180,E1 -18641.065,E2 -18641.065} C_VEL
LIN {X 0,Y 256.298,Z 156.558,A -85,B 0,C 180,E1 -18645.914,E2 -18645.914} C_VEL
LIN {X 0,Y 256.16,Z 156.575,A -85,B 0,C 180,E1 -18650.895,E2 -18650.895} C_VEL
LIN {X 0,Y 256.168,Z 156.573,A -85,B 0,C 180,E1 -18655.13,E2 -18655.13} C_VEL
LIN {X 0,Y 256.114,Z 156.58,A -85,B 0,C 180,E1 -18659.599,E2 -18659.599} C_VEL
LIN {X 0,Y 256.082,Z 156.584,A -85,B 0,C 180,E1 -18663.29,E2 -18663.29} C_VEL
LIN {X 0,Y 256.138,Z 156.576,A -85,B 0,C 180,E1 -18667.278,E2 -18667.278} C_VEL
LIN {X 0,Y 256.1,Z 156.582,A -85,B 0,C 180,E1 -18671.194,E2 -18671.194} C_VEL
LIN {X 0,Y 256.073,Z 156.586,A -85,B 0,C 180,E1 -18675.526,E2 -18675.526} C_VEL
LIN {X 0,Y 256.082,Z 156.584,A -85,B 0,C 180,E1 -18678.803,E2 -18678.803} C_VEL
LIN {X 0,Y 256.151,Z 156.573,A -85,B 0,C 180,E1 -18682.872,E2 -18682.872} C_VEL
LIN {X 0,Y 256.082,Z 156.584,A -85,B 0,C 180,E1 -18686.71,E2 -18686.71} C_VEL
LIN {X 0,Y 256.136,Z 156.579,A -85,B 0,C 180,E1 -18691.405,E2 -18691.405} C_VEL
LIN {X 0,Y 256.164,Z 156.576,A -85,B 0,C 180,E1 -18695.7,E2 -18695.7} C_VEL
LIN {X 0,Y 256.164,Z 156.575,A -85,B 0,C 180,E1 -18699.105,E2 -18699.105} C_VEL
LIN {X 0,Y 256.297,Z 156.557,A -85,B 0,C 180,E1 -18704.086,E2 -18704.086} C_VEL
LIN {X 0,Y 256.308,Z 156.557,A -85,B 0,C 180,E1 -18708.935,E2 -18708.935} C_VEL
LIN {X 0,Y 256.535,Z 156.528,A -85,B 0,C 180,E1 -18712.128,E2 -18712.128} C_VEL
LIN {X 0,Y 256.713,Z 156.506,A -85,B 0,C 180,E1 -18718.432,E2 -18718.432} C_VEL
LIN {X 0,Y 256.713,Z 156.505,A -85,B 0,C 180,E1 -18721.569,E2 -18721.569} C_VEL
LIN {X 0,Y 256.539,Z 156.527,A -85,B 0,C 180,E1 -18727.874,E2 -18727.874} C_VEL
LIN {X 0,Y 256.488,Z 156.531,A -85,B 0,C 180,E1 -18728.872,E2 -18728.872} C_VEL
LIN {X 0,Y 255.785,Z 156.623,A -85,B 0,C 180,E1 -18730.18,E2 -18730.18} C_VEL
LIN {X 0,Y 252.809,Z 156.992,A -85,B 0,C 180,E1 -18732.31,E2 -18732.31} C_VEL
LIN {X 0,Y 250.31,Z 157.303,A -85,B 0,C 180,E1 -18734.043,E2 -18734.043} C_VEL
LIN {X 0,Y 249.272,Z 157.433,A -85,B 0,C 180,E1 -18735.392,E2 -18735.392} C_VEL
LIN {X 0,Y 249.206,Z 157.441,A -85,B 0,C 180,E1 -18735.849,E2 -18735.849} C_VEL
LIN {X 0,Y 249.108,Z 157.452,A -85,B 0,C 180,E1 -18739.789,E2 -18739.789} C_VEL
LIN {X 0,Y 249.134,Z 157.45,A -85,B 0,C 180,E1 -18745.034,E2 -18745.034} C_VEL
LIN {X 0,Y 249.083,Z 157.454,A -85,B 0,C 180,E1 -18748.994,E2 -18748.994} C_VEL
LIN {X 0,Y 249.036,Z 157.464,A -85,B 0,C 180,E1 -18752.426,E2 -18752.426} C_VEL
LIN {X 0,Y 249.075,Z 157.457,A -85,B 0,C 180,E1 -18756.338,E2 -18756.338} C_VEL
LIN {X 0,Y 249.037,Z 157.463,A -85,B 0,C 180,E1 -18760.473,E2 -18760.473} C_VEL
LIN {X 0,Y 249.005,Z 157.463,A -85,B 0,C 180,E1 -18764.879,E2 -18764.879} C_VEL
LIN {X 0,Y 249.017,Z 157.466,A -85,B 0,C 180,E1 -18767.364,E2 -18767.364} C_VEL
LIN {X 0,Y 249.045,Z 157.464,A -85,B 0,C 180,E1 -18772.201,E2 -18772.201} C_VEL
LIN {X 0,Y 249.166,Z 157.527,A -85,B 0,C 180,E1 -18775.041,E2 -18775.041} C_VEL
LIN {X 0,Y 252.009,Z 171.603,A -85,B 0,C 180,E1 -18779.87,E2 -18779.87} C_VEL
LIN {X 0,Y 253.318,Z 178.783,A -85,B 0,C 180,E1 -18782.231,E2 -18782.231} C_VEL
LIN {X 0,Y 253.317,Z 179.657,A -85,B 0,C 180,E1 -18782.39,E2 -18782.39} C_VEL
LIN {X 0,Y 258.29,Z 230.714,A -85,B 0,C 180,E1 -18784.706,E2 -18784.706} C_VEL
LIN {X 0,Y 256.097,Z 289.404,A -85,B 0,C 180,E1 -18786.873,E2 -18786.873} C_VEL
LIN {X 0,Y 255.2,Z 302.322,A -85,B 0,C 180,E1 -18787.643,E2 -18787.643} C_VEL
LIN {X 0,Y 253.964,Z 314.962,A -85,B 0,C 180,E1 -18788.703,E2 -18788.703} C_VEL
LIN {X 0,Y 252.666,Z 327.196,A -85,B 0,C 180,E1 -18790.079,E2 -18790.079} C_VEL
LIN {X 0,Y 251.325,Z 338.304,A -85,B 0,C 180,E1 -18791.664,E2 -18791.664} C_VEL
LIN {X 0,Y 249.922,Z 349.365,A -85,B 0,C 180,E1 -18793.668,E2 -18793.668} C_VEL
LIN {X 0,Y 248.943,Z 358.404,A -85,B 0,C 180,E1 -18795.699,E2 -18795.699} C_VEL
LIN {X 0,Y 248.153,Z 365.838,A -85,B 0,C 180,E1 -18797.737,E2 -18797.737} C_VEL
LIN {X 0,Y 247.571,Z 373.081,A -85,B 0,C 180,E1 -18800.194,E2 -18800.194} C_VEL
LIN {X 0,Y 247.318,Z 378.8,A -85,B 0,C 180,E1 -18802.654,E2 -18802.654} C_VEL
LIN {X 0,Y 247.347,Z 383.227,A -85,B 0,C 180,E1 -18805.111,E2 -18805.111} C_VEL
LIN {X 0,Y 247.236,Z 385.503,A -85,B 0,C 180,E1 -18806.741,E2 -18806.741} C_VEL
LIN {X 0,Y 247.241,Z 387.302,A -85,B 0,C 180,E1 -18808.372,E2 -18808.372} C_VEL
LIN {X 0,Y 247.422,Z 388.617,A -85,B 0,C 180,E1 -18810.001,E2 -18810.001} C_VEL
LIN {X 0,Y 247.085,Z 389.913,A -85,B 0,C 180,E1 -18813.262,E2 -18813.262} C_VEL
LIN {X 0,Y 246.946,Z 389.883,A -85,B 0,C 180,E1 -18815.064,E2 -18815.064} C_VEL
LIN {X 0,Y 247.172,Z 388.674,A -85,B 0,C 180,E1 -18818.174,E2 -18818.174} C_VEL
LIN {X 0,Y 247.533,Z 387.468,A -85,B 0,C 180,E1 -18819.809,E2 -18819.809} C_VEL
LIN {X 0,Y 248.324,Z 384.851,A -85,B 0,C 180,E1 -18822.256,E2 -18822.256} C_VEL
LIN {X 0,Y 249.684,Z 381.251,A -85,B 0,C 180,E1 -18824.675,E2 -18824.675} C_VEL
LIN {X 0,Y 251.537,Z 376.582,A -85,B 0,C 180,E1 -18827.061,E2 -18827.061} C_VEL
LIN {X 0,Y 254.053,Z 369.599,A -85,B 0,C 180,E1 -18829.852,E2 -18829.852} C_VEL
LIN {X 0,Y 256.878,Z 362.299,A -85,B 0,C 180,E1 -18832.098,E2 -18832.098} C_VEL
LIN {X 0,Y 260.181,Z 353.207,A -85,B 0,C 180,E1 -18834.327,E2 -18834.327} C_VEL
LIN {X 0,Y 263.725,Z 342.937,A -85,B 0,C 180,E1 -18836.299,E2 -18836.299} C_VEL
LIN {X 0,Y 267.248,Z 331.514,A -85,B 0,C 180,E1 -18838.039,E2 -18838.039} C_VEL
LIN {X 0,Y 270.297,Z 320.243,A -85,B 0,C 180,E1 -18839.392,E2 -18839.392} C_VEL
LIN {X 0,Y 273.522,Z 306.576,A -85,B 0,C 180,E1 -18840.603,E2 -18840.603} C_VEL
LIN {X 0,Y 275.757,Z 294.643,A -85,B 0,C 180,E1 -18841.391,E2 -18841.391} C_VEL
LIN {X 0,Y 277.563,Z 280.342,A -85,B 0,C 180,E1 -18842.069,E2 -18842.069} C_VEL
LIN {X 0,Y 281.36,Z 235.911,A -85,B 0,C 180,E1 -18843.685,E2 -18843.685} C_VEL
LIN {X 0,Y 280.163,Z 221.17,A -85,B 0,C 180,E1 -18844.828,E2 -18844.828} C_VEL
LIN {X 0,Y 279.316,Z 214.852,A -85,B 0,C 180,E1 -18845.421,E2 -18845.421} C_VEL
LIN {X 0,Y 275.962,Z 206.746,A -85,B 0,C 180,E1 -18846.871,E2 -18846.871} C_VEL
